// TwinCAT 3 PLC project tesimplc
// ProgramVersion: 3.1.0.8
// libraries:
//   Tc2_ControllerToolbox, * (Beckhoff Automation GmbH)
//   Tc2_Math, * (Beckhoff Automation GmbH)
//   Tc2_ModbusSrv, * (Beckhoff Automation GmbH)
//   Tc2_Standard, * (Beckhoff Automation GmbH)
//   Tc2_System, * (Beckhoff Automation GmbH)
//   Tc2_TcpIp, * (Beckhoff Automation GmbH)
//   Tc2_Utilities, * (Beckhoff Automation GmbH)
//   Tc3_Interfaces, * (Beckhoff Automation GmbH)
//   Tc3_Module, * (Beckhoff Automation GmbH)
// project tree:
//   DUTs/ MODBUS_DATA_MAP.TcDUT, XMEAS_IDX.TcDUT, XMEAS_IO_IDX.TcDUT, XMEAS_MBS_IDX.TcDUT, XMV_IDX.TcDUT, XMV_IO_IDX.TcDUT
//   funcs/ adc_to_float_pv.TcPOU (not stored), pv_float_to_dac.TcPOU
//   / GlobalTextList.TcGTLO, MainTask.TcTTO, Visualization Manager.TcVMO (not stored), VISU_TASK.TcTTO
//   GVLs/ GVL_NAMES.TcGVL, G_ICAL.TcGVL, G_IO.TcGVL, G_PARAMS.TcGVL
//   POUs/FBModbus/ FB_mb_to_val.TcPOU, FB_ModbusPoll.TcPOU, FB_ReadModbus.TcPOU, FB_HexStringToReal.TcPOU
//   POUs/FBUtils/ FB_CSV_Writer.TcPOU, FB_LFSR.TcPOU, FB_recursiveFilter.TcPOU
//   POUs/FB_Networks/ FB_NoNet.TcPOU
//   POUs/FB_Networks/iMesh/ FB_3eTI_iMesh_Base.TcPOU, FB_3eTI_iMesh_Cal.TcPOU, FB_3eTI_iMesh_GasSensor.TcPOU, FB_3eTI_iMesh_LFSR.TcPOU, FB_3eTI_iMesh_TESIM.TcPOU, FB_3eTI_TestSignals.TcPOU
//   POUs/FB_Networks/PCOneLink/ FB_PC_LFSR.TcPOU, FB_PC_OneLink_Base.TcPOU, FB_PC_OneLink_Cal.TcPOU, FB_PC_OneLink_GasSensor.TcPOU, FB_PC_OneLink_TESIM.TcPOU, FB_PC_OneLink_TestSignals.TcPOU
//   POUs/FB_Networks/Yokogawa/ FB_Yokogawa_LFSR.TcPOU, FB_Yokogawa_TestSignals.TcPOU, FB_Yokogawa_Base.TcPOU, FB_Yokogawa_GasSensor.TcPOU
//   POUs/ MAIN_oo.TcPOU
//   VISUs/ ImagePool.TcIPO (not stored), TankView.TcVIS, TESimView.TcPOU
//   zzArchive/ MAIN_wsn.TcPOU
// real-time tasks:
//   TASK MainTask: cycle T#10ms, priority 1, ADS port 350
//   TASK VISU_TASK: cycle T#100000us, priority 30, ADS port 351
// I/O:
//   DEVICE Device 1 (EtherCAT), AmsNetId 5.20.215.224.2.1
//     Term 1 (EK1200) [EK1200-5000 EtherCAT Power supply (2A E-Bus)]
//       Term 2 (EL3058) [EL3058 8Ch. Ana. Input 4-20mA]
//       Term 3 (EL4028) [EL4028 8Ch. Ana. Output 4-20mA, 12bit]
//       Term 4 (EL1808) [EL1808 8Ch. Dig. Input 24V, 3ms]
//       Term 5 (EL2808) [EL2808 8Ch. Dig. Output 24V, 0.5A]
//       Term 6 (EL3068) [EL3068 8Ch. Ana. Input 0-10V]
//       Term 7 (EL4008) [EL4008 8Ch. Ana. Output 0-10V, 12bit]
//       Term 8 (EL9011) [EL9011 End Terminal]
// variable links:
//   tesimplc/tesimplc Instance <-> Device 1 (EtherCAT)/Term 1 (EK1200)/Term 2 (EL3058)
//     MainTask Inputs/G_IO.XMEAS_IO_IIN[{1..4}] <-> AI Standard Channel {1..4}/Value  (4 links)
//     MainTask Inputs/G_IO.XMV_IO_IIN[{1..4}] <-> AI Standard Channel {5..8}/Value  (4 links)
//   tesimplc/tesimplc Instance <-> Device 1 (EtherCAT)/Term 1 (EK1200)/Term 3 (EL4028)
//     MainTask Outputs/G_IO.XMEAS_IO_IOUT[{1..4}] <-> AO Outputs Channel {1..4}/Analog output  (4 links)
//     MainTask Outputs/G_IO.XMV_IO_IOUT[{1..4}] <-> AO Outputs Channel {5..8}/Analog output  (4 links)
//   tesimplc/tesimplc Instance <-> Device 1 (EtherCAT)/Term 1 (EK1200)/Term 7 (EL4008)
//     MainTask Outputs/G_IO.XMEAS_IO_VOUT[{1..8}] <-> AO Outputs Channel {1..8}/Analog output  (8 links)

CONFIGURATION tesimplc
    RESOURCE PLC ON TwinCAT3
        TASK MainTask(INTERVAL := T#10ms, PRIORITY := 1);
        TASK VISU_TASK(INTERVAL := T#100000us, PRIORITY := 30);
        PROGRAM MAIN_oo WITH MainTask : MAIN_oo;
        PROGRAM VisuElems_Visu_Prg WITH VISU_TASK : VisuElems.Visu_Prg;
    END_RESOURCE
END_CONFIGURATION

// ---- DUTs/MODBUS_DATA_MAP.TcDUT
TYPE MODBUS_DATA_MAP :
STRUCT
	_ipAddress : STRING;
	_startAddress : WORD;
END_STRUCT
END_TYPE

// ---- DUTs/XMEAS_IDX.TcDUT
TYPE XMEAS_IDX:	
	( 
		A_FLOW			:=1,
		D_FLOW			:=2,
		E_FLOW			:=3,
		AC_FLOW			:=4,
		P_REACTOR		:=7,
		L_REACTOR		:=8,
		T_REACTOR		:=9,
		L_SEPARATOR		:=12,
		L_STRIPPER		:=15
	);
END_TYPE

// ---- DUTs/XMEAS_IO_IDX.TcDUT
TYPE XMEAS_IO_IDX :
	( 
		A_FLOW			:=1,
		D_FLOW			:=2,
		E_FLOW			:=3,
		P_REACTOR		:=4,
		AC_FLOW			:=4
	);
END_TYPE

// ---- DUTs/XMEAS_MBS_IDX.TcDUT
TYPE XMEAS_MBS_IDX :
(
	A_FLOW			:=1,
	D_FLOW			:=2,
	E_FLOW			:=3,
	P_REACTOR		:=4,
	AC_FLOW			:=4
);
END_TYPE

// ---- DUTs/XMV_IDX.TcDUT
TYPE XMV_IDX :
(
	D_FLOW_VALVE			:=1,
	E_FLOW_VALVE			:=2,	
	A_FLOW_VALVE			:=3,
	REACTOR_CWFV			:=10
);
END_TYPE

// ---- DUTs/XMV_IO_IDX.TcDUT
TYPE XMV_IO_IDX :
(
	D_FLOW_VALVE			:=1,
	E_FLOW_VALVE			:=2,	
	A_FLOW_VALVE			:=3,
	REACTOR_CWFV			:=4
);
END_TYPE

// ---- GVLs/GVL_NAMES.TcGVL
VAR_GLOBAL
	xmv_names: ARRAY[1..12] OF STRING := [
		'D Feed',
		'E Feed',
		'A Feed',
		'A+C Feed',
		'Recycle Valve',
		'Purge Valve',
		'Separator Valve',
		'Stripper Valve',
		'Steam valve',
		'Reactor Coolant',
		'Condenser Coolant',
		'Agitator Speed' ];

	xmeas_names: ARRAY[1..41] OF STRING := [
		'A Feed (kscmh)',
		'D Feed (kg/hr)',
		'E Feed (kg/hr)',
		'A+C Feed (kscmh)',
		'Recycle Flow (kscmh)',
		'Reactor Feed (kscmh)',
		'Reactor Pressure (kPa)',
		'Reactor Level (%)',
		'Reactor Temp. (°C)',
		'Purge Rate (kscmh)',
		'Sep Temp. (°C)',
		'Sep Level (%)',
		'Sep Pressure (kPa)',
		'Sep Underflow (m³/hr)',
		'Stripper Level (%)',
		'Stripper Pressure (kPa)',
		'Stripper Underflow (m³/hr)',
		'Stripper Temp. (°C)',
		'Steam Flow (kg/hr)',
		'Compressor Work (kW)',
		'React. Cool. Temp. (°C)',
		'Cond. Cool. Temp. (°C)',
		'Feed A (mole %)',
		'Feed B (mole %)',
		'Feed C (mole %)',
		'Feed D (mole %)',
		'Feed E (mole %)',
		'Feed F (mole %)',
		'Purge     % A (mole %)',
		'Purge     % B (mole %)',
		'Purge     % C (mole %)',
		'Purge     % D (mole %)',
		'Purge     % E (mole %)',
		'Purge     % F (mole %)',
		'Purge     % G (mole %)',
		'Purge     % H (mole %)',
		'Product D (mole %)',
		'Product E (mole %)',
		'Product F (mole %)',
		'Product G (mole %)',
		'Product H (mole %)' ];
END_VAR

// ---- GVLs/G_ICAL.TcGVL
VAR_GLOBAL
	
	// represents the net DC offset compensation multiplier
	XMEAS_ILOOP_CAL	: ARRAY[1..4] OF LREAL	:= 
				[
					// XMEAS tx-rx path
					-39, // A flow
					-9, // D flow
					8, // E flow
					4  // Reactor pressure
				];		
				
	XMV_ILOOP_CAL	: ARRAY[1..4] OF LREAL	:= 
				[
					// XMV tx-rx path
					-11, 	// D valve
					-11, 	// E valve
					15, 	// A valve
					-1	 	// RCW Valve
				];					
END_VAR

// ---- GVLs/G_IO.TcGVL
VAR_GLOBAL CONSTANT
	
END_VAR

VAR_GLOBAL
	
	// specify network type
	// 100 					: ISA110.11a iMesh calibration
	// 101 					: ISA110.11a iMesh TESIM
	// 102 					: ISA110.11a iMesh test signals
	// 110					: ISA100.11a iMesh PN Sequence generation
	
	// 200 					: PhoenixContact calibration
	// 201					: PhoenixContact TESIM
	// 202					: PhoenixContact test signals
	// 210					: ISA100.11a PC OneLink PN Sequence generation
	
	NET_TYPE				:	DINT := 0;
	GO						:	BOOL := FALSE;
	MODE					:	UINT := 1;
	
	// operating time
	OPTIME					:	LREAL := 0.0;
	
	// for the current-based control solutions
	XMEAS_IO_IOUT	AT %Q*		:	ARRAY[1..4] OF INT;
	XMEAS_IO_IIN	AT %I*		:	ARRAY[1..4] OF INT;
	XMV_IO_IOUT		AT %Q*		:	ARRAY[1..4] OF INT;
	XMV_IO_IIN		AT %I*		:	ARRAY[1..4] OF INT;
	
	// for the voltage-based control solutions
	XMEAS_IO_VOUT 	AT %Q*		:	ARRAY[1..8] OF INT;
	
	// XMEAS reported by tesim
	XMEAS						:	ARRAY[1..41] OF LREAL;
	XMEAS_RX					:	ARRAY[1..41] OF LREAL;
	
	// XMEAS seen by the network
	MBS_XMEAS_RAW				:	ARRAY[1..4] OF REAL;
	MBS_XMEAS					:	ARRAY[1..4] OF REAL;
	MBS_XMEAS_CAL_OFFSET		:	ARRAY[1..4] OF REAL := [0.0215, 0.0175, 0.0195, 0.0216];

	// XMV values reported by tesim
	XMV							:	ARRAY[1..12] OF LREAL;
	XMV_RX						:	ARRAY[1..12] OF LREAL;
	
	// XMV seen by the network
	//NET_XMV_RAW						:	ARRAY[1..4] OF LREAL;
	NET_XMV							:	ARRAY[1..4] OF REAL;
	
	// setpoints
	PROD_RATE					:	LREAL;
	P_REACTOR					:	LREAL;
	L_REACTOR					:	LREAL;
	T_REACTOR					:	LREAL;
	PCT_G_SP					:	LREAL;
	L_SEPARATOR					:	LREAL;
	L_STRIPPER					:	LREAL;
	
	// filtered (smoothed) values
	P_REACTOR_SM					:	LREAL;
	
	// production metrics
	COST						:	LREAL :=0.0;
	PctG						:	LREAL :=0.0;
	
	// disturbances as set in tesim
	IDV							:	ARRAY[1..20] OF DINT;
	
	// shutdown indicator
	SD_FLAG						: 	BOOL	:= FALSE;
	
END_VAR

// ---- GVLs/G_PARAMS.TcGVL
VAR_GLOBAL
	IOUT_WD_MAX	:	INT		:=32767;
	IOUT_WD_MIN	:	INT		:=0;
	VOUT_WD_MAX	:	INT		:=32767;
	VOUT_WD_MIN	:	INT		:=0;
	
	// XMEAS RANGES
	A_FLOW_MAX 		:	LREAL	:=10.0;
	D_FLOW_MAX		:	LREAL	:=7500.0;
	E_FLOW_MAX		:	LREAL	:=7500.0;
	AC_FLOW_MAX		:	LREAL	:=50.0;
	P_REACTOR_MAX	:	LREAL	:=3000.0;
	
	A_FLOW_MIN 		:	LREAL	:=0.0;
	D_FLOW_MIN		:	LREAL	:=0.0;
	E_FLOW_MIN		:	LREAL	:=0.0;
	AC_FLOW_MIN		:	LREAL	:=0.0;
	P_REACTOR_MIN	:	LREAL	:=0.0;
	
	// XMV RANGES
	A_FLOW_VALVE_MAX	: LREAL	:=100.0;
	D_FLOW_VALVE_MAX	: LREAL	:=100.0;
	E_FLOW_VALVE_MAX	: LREAL	:=100.0;
	REACTOR_CWFV_MAX	: LREAL	:=100.0;
	
	A_FLOW_VALVE_MIN	: LREAL			:=0.0;
	D_FLOW_VALVE_MIN	: LREAL			:=0.0;
	E_FLOW_VALVE_MIN	: LREAL			:=0.0;
	REACTOR_CWFV_MIN	: LREAL			:=0.0;
	
	// Device limits
	VOUT_MAX		:	LREAL	:=10.0;
	VOUT_MIN		:	LREAL	:=0.0;
	IOUT_MAX		:	LREAL	:=20.0;
	IOUT_MIN		:	LREAL	:=4.0;
	

END_VAR

// ---- POUs/MAIN_oo.TcPOU
PROGRAM MAIN_oo
VAR
	
	// network interface/simulator function blocks
	netiMeshCal				:FB_3eTI_iMesh_Cal;
	netiMeshTESIM			:FB_3eTI_iMesh_TESIM;
	netiMeshTestSignals		:FB_3eTI_TestSignals;
	netiMeshGasSensor		:FB_3eTI_iMesh_GasSensor;
	netiMeshLFSR			:FB_3eTI_iMesh_LFSR;
	
	netPCCal				:FB_PC_OneLink_Cal;
	netPCTESIM				:FB_PC_OneLink_TESIM;
	netPCTestSignals		:FB_PC_OneLink_TestSignals;
	netPCGasSensor			:FB_PC_OneLink_GasSensor;
	netPC_LFSR				:FB_PC_LFSR;
	
	// yokogawa signals
	netYokoTestSignals		:FB_Yokogawa_TestSignals;
	netYokoLFSR				:FB_Yokogawa_LFSR;
	netYokoGasSensor		:FB_Yokogawa_GasSensor;

	netNoNet				:FB_NoNet;
	
END_VAR



CASE NET_TYPE OF 
	100:
	netiMeshCal();
	101:
	netiMeshTESIM();
	102:
	netiMeshTestSignals();
	103:
	netiMeshGasSensor();
	110:
	netiMeshLFSR();
	
	200:
	netPCCal();
	201:
	netPCTESIM();
	202:
	netPCTestSignals();
	203:
	netPCGasSensor();	
	210:
	netPC_LFSR();
	
	300:
	301:
	302:
	netYokoTestSignals();
	303:
	netYokoGasSensor();
	310:
	netYokoLFSR();
	
	
ELSE
	netnoNet();
	
END_CASE

END_PROGRAM

// ---- POUs/FB_Networks/iMesh/FB_3eTI_iMesh_Cal.TcPOU
FUNCTION_BLOCK FB_3eTI_iMesh_Cal EXTENDS FB_3eTI_TestSignals
VAR_INPUT
END_VAR
VAR_OUTPUT
END_VAR
VAR
		//common calibration variables
	cal_tm 			:	TIME := T#20S;
	cal_tm_task 	:	TIME := T#100MS;
	cal_emode : E_CTRL_MODE := eCTRL_MODE_ACTIVE;
	cal_override	: BOOL	:= TRUE;
	cal_pv_mbs: ARRAY[1..4] OF LREAL := [0.0,0.0,0.0,0.0];
	cal_pv: ARRAY[1..4] OF LREAL := [0.0,0.0,0.0,0.0];
		
	// moving average
	cal_mva_work:	ARRAY[1..4] OF ARRAY[1..cal_mva_nWorkArray_SIZEOF] OF LREAL;
	cal_mva_st	:   ARRAY[1..4] OF ST_CTRL_MOVING_AVERAGE_PARAMS := [
		(	tTaskCycleTime:=cal_tm_task, 
			tCtrlCycleTime:=cal_tm,
			nSamplesToFilter:=cal_mva_nSamplesToFilter,
			nWorkArray_SIZEOF:=cal_mva_nWorkArray_SIZEOF),
		(	tTaskCycleTime:=cal_tm_task, 
			tCtrlCycleTime:=cal_tm,
			nSamplesToFilter:=cal_mva_nSamplesToFilter,
			nWorkArray_SIZEOF:=cal_mva_nWorkArray_SIZEOF),
		(	tTaskCycleTime:=cal_tm_task, 
			tCtrlCycleTime:=cal_tm,
			nSamplesToFilter:=cal_mva_nSamplesToFilter,
			nWorkArray_SIZEOF:=cal_mva_nWorkArray_SIZEOF),
		(	tTaskCycleTime:=cal_tm_task, 
			tCtrlCycleTime:=cal_tm,
			nSamplesToFilter:=cal_mva_nSamplesToFilter,
			nWorkArray_SIZEOF:=cal_mva_nWorkArray_SIZEOF)
	];
	fb_cal_mva	:	ARRAY[1..4] OF FB_CTRL_MOVING_AVERAGE := [ 
		(eMode:=cal_emode), 
		(eMode:=cal_emode), 
		(eMode:=cal_emode), 
		(eMode:=cal_emode)];
	cal_mva_mbs :	ARRAY[1..4] OF LREAL;

	// more common cal vars		
	cal_10v_dcoffset: ARRAY[1..4] OF LREAL;
	cal_ii: INT;
	cal_diff: ARRAY[1..4] OF LREAL;
	cal_frac: ARRAY[1..4] OF LREAL;
	
END_VAR
VAR CONSTANT
	cal_mva_nSamplesToFilter : UINT := 40;
	cal_mva_nWorkArray_SIZEOF: UINT := 400;
END_VAR


// call the base class to query test signal values
SUPER^();

// CALIBRATION SECTION
IF cal_override THEN
	FOR cal_ii := 1 TO 4 DO
		CASE cal_ii OF
			1:
			G_IO.XMEAS[XMEAS_IDX.A_FLOW]:=0.5;
			2:
			G_IO.XMEAS[XMEAS_IDX.D_FLOW] := 1500;
			3:
			G_IO.XMEAS[XMEAS_IDX.E_FLOW] := 1500;
			4:
			G_IO.XMEAS[XMEAS_IDX.AC_FLOW] := 2500;
		END_CASE
	END_FOR
END_IF
IF cal_emode=eCTRL_MODE_ACTIVE THEN
	FOR cal_ii := 1 TO 4 DO
		CASE cal_ii OF
			1:
			cal_pv_mbs[cal_ii] := G_IO.MBS_XMEAS[XMEAS_MBS_IDX.A_FLOW];
			cal_pv[cal_ii] := G_IO.XMEAS[XMEAS_IDX.A_FLOW];
			2:
			cal_pv_mbs[cal_ii] := G_IO.MBS_XMEAS[XMEAS_MBS_IDX.D_FLOW];
			cal_pv[cal_ii] := G_IO.XMEAS[XMEAS_IDX.D_FLOW];
			3:
			cal_pv_mbs[cal_ii] := G_IO.MBS_XMEAS[XMEAS_MBS_IDX.E_FLOW];
			cal_pv[cal_ii] := G_IO.XMEAS[XMEAS_IDX.E_FLOW];
			4:
			cal_pv_mbs[cal_ii] := G_IO.MBS_XMEAS[XMEAS_MBS_IDX.AC_FLOW];
			cal_pv[cal_ii] := G_IO.XMEAS[XMEAS_IDX.AC_FLOW];
		END_CASE
	
		// calculate moving average
		cal_mva_st[cal_ii].pWorkArray_ADR	:= ADR(cal_mva_work[cal_ii]);
		fb_cal_mva[cal_ii].fIn := cal_pv_mbs[cal_ii];
		fb_cal_mva[cal_ii](stParams:=cal_mva_st[cal_ii], eMode:=cal_emode);
		cal_mva_mbs[cal_ii] := fb_cal_mva[cal_ii].fOut;	
		
		// calculate dc offset
		IF ABS(cal_pv[cal_ii]) > 0.0 THEN
			cal_diff[cal_ii]:=cal_mva_mbs[cal_ii]-cal_pv[cal_ii];
			cal_frac[cal_ii]:=cal_diff[cal_ii]/cal_pv[cal_ii];
			cal_10v_dcoffset[cal_ii] := 10.0*cal_frac[cal_ii];
		END_IF
		
	END_FOR	
END_IF

END_FUNCTION_BLOCK

// ---- POUs/FB_Networks/iMesh/FB_3eTI_TestSignals.TcPOU
FUNCTION_BLOCK FB_3eTI_TestSignals EXTENDS FB_3eTI_iMesh_Base
VAR_INPUT
END_VAR
VAR_OUTPUT
END_VAR
VAR
END_VAR


G_PARAMS.A_FLOW_MAX 		:=10.0;
G_PARAMS.D_FLOW_MAX			:=10.0;
G_PARAMS.E_FLOW_MAX			:=10.0;
G_PARAMS.AC_FLOW_MAX		:=10.0;

G_PARAMS.A_FLOW_MIN 		:=0.0;
G_PARAMS.D_FLOW_MIN			:=0.0;
G_PARAMS.E_FLOW_MIN			:=0.0;
G_PARAMS.AC_FLOW_MIN		:=0.0;

// execute the signal conversion
SUPER^();

END_FUNCTION_BLOCK

// ---- POUs/FB_Networks/iMesh/FB_3eTI_iMesh_Base.TcPOU
FUNCTION_BLOCK FB_3eTI_iMesh_Base
VAR_INPUT
	
	// THIS IS FOR THE ISA100.11A GATEWAY
	mbAddrs : ARRAY[1..4] OF MODBUS_DATA_MAP :=  [ 
			(_ipAddress := '192.168.254.253', _startAddress:= 6), 
			(_ipAddress := '192.168.254.253', _startAddress:= 18),
			(_ipAddress := '192.168.254.253', _startAddress:= 30),
			(_ipAddress := '192.168.254.253', _startAddress:= 42)
		];
		
END_VAR

VAR
	fbReadMB 	: FB_ReadModbus;
	ii			: INT:=0;
END_VAR

VAR_OUTPUT
END_VAR

VAR
END_VAR

//
// BEGIN PRODUCE THE DATA
//
// XMEAS values will come from the external TESIM program using ADS

// VOLTAGES
XMEAS_IO_VOUT[XMEAS_IO_IDX.A_FLOW]		:= pv_float_to_dac(pv:=XMEAS[XMEAS_IDX.A_FLOW],		pv_max:=G_PARAMS.A_FLOW_MAX, pv_min:=G_PARAMS.A_FLOW_MIN, dac_max:=VOUT_WD_MAX, dac_min:=0);
XMEAS_IO_VOUT[XMEAS_IO_IDX.D_FLOW]		:= pv_float_to_dac(pv:=XMEAS[XMEAS_IDX.D_FLOW],		pv_max:=G_PARAMS.D_FLOW_MAX, pv_min:=G_PARAMS.D_FLOW_MIN, dac_max:=VOUT_WD_MAX, dac_min:=0);
XMEAS_IO_VOUT[XMEAS_IO_IDX.E_FLOW]		:= pv_float_to_dac(pv:=XMEAS[XMEAS_IDX.E_FLOW],		pv_max:=G_PARAMS.E_FLOW_MAX, pv_min:=G_PARAMS.E_FLOW_MIN, dac_max:=VOUT_WD_MAX, dac_min:=0);
XMEAS_IO_VOUT[XMEAS_IO_IDX.AC_FLOW]	:= pv_float_to_dac(pv:=XMEAS[XMEAS_IDX.AC_FLOW],	pv_max:=G_PARAMS.AC_FLOW_MAX, pv_min:=G_PARAMS.AC_FLOW_MIN, dac_max:=VOUT_WD_MAX, dac_min:=0);

//
// BEGIN MODBUS POLLING SEGMENT from the GATEWAY
//
fbReadMB(n:=4, addrs := ADR(mbAddrs) );

// poll modbus registers
G_IO.MBS_XMEAS_RAW[XMEAS_MBS_IDX.A_FLOW] := fbReadMB.registerValues[XMEAS_MBS_IDX.A_FLOW] + MBS_XMEAS_CAL_OFFSET[1];
G_IO.MBS_XMEAS_RAW[XMEAS_MBS_IDX.D_FLOW] := fbReadMB.registerValues[XMEAS_MBS_IDX.D_FLOW]+ MBS_XMEAS_CAL_OFFSET[2];
G_IO.MBS_XMEAS_RAW[XMEAS_MBS_IDX.E_FLOW] := fbReadMB.registerValues[XMEAS_MBS_IDX.E_FLOW] + MBS_XMEAS_CAL_OFFSET[3];
G_IO.MBS_XMEAS_RAW[XMEAS_MBS_IDX.AC_FLOW] := fbReadMB.registerValues[XMEAS_MBS_IDX.AC_FLOW] + MBS_XMEAS_CAL_OFFSET[4];

// convert raw modbus signals to process signals
G_IO.MBS_XMEAS[XMEAS_MBS_IDX.A_FLOW]	:=	LREAL_TO_REAL(adc_to_float_pv(G_IO.MBS_XMEAS_RAW[XMEAS_MBS_IDX.A_FLOW],		pv_max:=G_PARAMS.A_FLOW_MAX, 		pv_min:=G_PARAMS.A_FLOW_MIN, 	i_max:=G_PARAMS.VOUT_MAX, i_min:=G_PARAMS.VOUT_MIN));
G_IO.MBS_XMEAS[XMEAS_MBS_IDX.D_FLOW]	:=	LREAL_TO_REAL(adc_to_float_pv(G_IO.MBS_XMEAS_RAW[XMEAS_MBS_IDX.D_FLOW],		pv_max:=G_PARAMS.D_FLOW_MAX, 		pv_min:=G_PARAMS.D_FLOW_MIN, 	i_max:=G_PARAMS.VOUT_MAX, i_min:=G_PARAMS.VOUT_MIN));
G_IO.MBS_XMEAS[XMEAS_MBS_IDX.E_FLOW]	:=	LREAL_TO_REAL(adc_to_float_pv(G_IO.MBS_XMEAS_RAW[XMEAS_MBS_IDX.E_FLOW],		pv_max:=G_PARAMS.E_FLOW_MAX, 		pv_min:=G_PARAMS.E_FLOW_MIN, 	i_max:=G_PARAMS.VOUT_MAX, i_min:=G_PARAMS.VOUT_MIN));
G_IO.MBS_XMEAS[XMEAS_MBS_IDX.AC_FLOW]	:=	LREAL_TO_REAL(adc_to_float_pv(G_IO.MBS_XMEAS_RAW[XMEAS_MBS_IDX.AC_FLOW],	pv_max:=G_PARAMS.AC_FLOW_MAX, 	pv_min:=G_PARAMS.AC_FLOW_MIN, i_max:=G_PARAMS.VOUT_MAX, i_min:=G_PARAMS.VOUT_MIN));

// capture the received state of XMEAS
FOR ii := 1 TO 41 DO
	XMEAS_RX[ii]:=XMEAS[ii];
END_FOR
XMEAS_RX[XMEAS_IDX.A_FLOW] := G_IO.MBS_XMEAS[XMEAS_MBS_IDX.A_FLOW];
XMEAS_RX[XMEAS_IDX.D_FLOW] := G_IO.MBS_XMEAS[XMEAS_MBS_IDX.D_FLOW];
XMEAS_RX[XMEAS_IDX.E_FLOW] := G_IO.MBS_XMEAS[XMEAS_MBS_IDX.E_FLOW];
XMEAS_RX[XMEAS_IDX.AC_FLOW] := G_IO.MBS_XMEAS[XMEAS_MBS_IDX.AC_FLOW];

// capture the received state of XMV
FOR ii := 1 TO 12 DO
	XMV_RX[ii]:=XMV[ii];
END_FOR

//
// END MODBUS POLLING SEGMENT from the GATEWAY
//

END_FUNCTION_BLOCK

// ---- POUs/FBModbus/FB_ReadModbus.TcPOU
FUNCTION_BLOCK FB_ReadModbus

VAR_INPUT
	n			: INT; 	// number of modbus clients
	addrs 		: POINTER TO ARRAY[1..50] OF MODBUS_DATA_MAP;
	intervalToSampleData : TIME := T#1S; 	//modbus update rate (lower rate = more disk usage) default : 5 seconds
END_VAR

VAR_OUTPUT
	
	// input register values
	registerValues : ARRAY[0..50] OF REAL;
END_VAR

VAR
	addr: MODBUS_DATA_MAP;
	mb	: ARRAY[1..50] OF FB_ModbusPoll;
	
	//holds how many readings have been taken from initial download
	numberOfReadingsTaken : INT;

	ii: INT;
END_VAR


FOR ii:=1 TO n DO
	addr := addrs^[ii];
	mb[ii].ipAd := addr._ipAddress;
	mb[ii].startAddr := addr._startAddress;
	mb[ii](value => registerValues[ii]);
END_FOR

END_FUNCTION_BLOCK

// ---- POUs/FBModbus/FB_ModbusPoll.TcPOU
FUNCTION_BLOCK FB_ModbusPoll

VAR_INPUT
	ipAd : STRING; // the ip address of the modbus server
	startAddr : WORD; // the start address
END_VAR

VAR_OUTPUT
	value : REAL; //the modbus data
END_VAR

VAR
	dataStr :STRING;
	bModbusTick : BOOL;
	fbReadRegs : FB_MBReadInputRegs;
	converter : FB_HexStringToReal;
	arr : ARRAY [0..2] OF WORD;
END_VAR

//setup the modbus block
fbReadRegs.sIPAddr := ipAd; //gateway ip
fbReadRegs.nTCPPort := MODBUS_TCP_PORT; //502
fbReadRegs.nUnitID := 16#FF; //255
fbReadRegs.nQuantity := 3; //3 words
fbReadRegs.tTimeout := T#5S; //30 sec timout
fbReadRegs.nMBAddr := startAddr;
fbReadRegs.cbLength := 6;//nQuantity*2
fbReadRegs.pDestAddr := ADR(arr); //the pointer to the array

//the rising edge of the input negate the tick to create  a rising input of change :)
fbReadRegs.bExecute := (bModbusTick := NOT bModbusTick);
//fbReadRegs.bExecute := (bModbusTick := TRUE); 

//uppercase(convert first number to hex + convert second number to hex)
dataStr := F_TOUCase(CONCAT(WORD_TO_HEXSTR(arr[1],4,TRUE),WORD_TO_HEXSTR(arr[2],4,TRUE))); 
fbReadRegs();

//use converter to convert last 2 words to a fp value
converter(str := dataStr, out => value);

END_FUNCTION_BLOCK

// ---- POUs/FBModbus/FB_HexStringToReal.TcPOU
FUNCTION_BLOCK FB_HexStringToReal
VAR_INPUT
	str :STRING;
END_VAR
VAR_OUTPUT
	out : REAL;
END_VAR
VAR
holdStr : STRING := '';
binStr : STRING := '';
bin : STRING := '';	
sExponent : INT := 1;
expVal : INT;
sMantissa : STRING;
i :INT :=0;
ar : ARRAY[0..23] OF STRING;
significand : REAL;
decVal : REAL ;

mySExponent:INT;
myEVal:REAL;
myOut:REAL;
END_VAR

//converts the hex string to binary
FOR i :=1 TO 8 BY 1 DO
	holdStr := MID(str,1,i);
	
	IF holdStr = '0' THEN
		bin := '0000';
	ELSIF holdStr = '1' THEN
		bin := '0001';
	ELSIF holdStr = '2' THEN
		bin := '0010';
	ELSIF holdStr = '3' THEN
		bin := '0011';
	ELSIF holdStr = '4' THEN
		bin := '0100';
	ELSIF holdStr = '5' THEN
		bin := '0101';
	ELSIF holdStr = '6' THEN
		bin := '0110';
	ELSIF holdStr = '7' THEN
		bin := '0111';
	ELSIF holdStr = '8' THEN
		bin := '1000';
	ELSIF holdStr = '9' THEN
		bin := '1001';
	ELSIF holdStr = 'A' THEN
		bin := '1010';
	ELSIF holdStr = 'B' THEN
		bin := '1011';
	ELSIF holdStr = 'C' THEN
		bin := '1100';
	ELSIF holdStr = 'D' THEN
		bin := '1101';
	ELSIF holdStr = 'E' THEN
		bin := '1110';
	ELSIF holdStr = 'F' THEN
		bin := '1111';
	END_IF
	
	binStr := CONCAT(binStr,bin);
		
END_FOR

//takes half of the string
binStr := RIGHT(binStr,32);

//gets rid of the sign bit bc i am assuming that it is always positive
binStr := DELETE(binStr,1,1);

//convert the first 8 bits to get the exponent value and subtract 127
sExponent := STRING_TO_INT(CONCAT('2#',LEFT(binStr,8))) - 127;

//get remaining 23 mantissa bits
sMantissa := MID(binStr,23,9);

//values to divide by
decVal := 0.5;

//mantissa value
significand := 0;

//store mantissa bits in array
FOR i := 0 TO 23 BY 1 DO
	ar[i] := MID(sMantissa,1,i);
END_FOR

//get the significand by multiplying current bit by decVal then halve the decVal
FOR i:= 1 TO 23 BY 1 DO
	significand := significand + (STRING_TO_INT(ar[i])*decVal);
	decVal := decVal/2.0;
END_FOR

//manually generate the power of 2
expVal := 2;
FOR i:= 0 TO sExponent-2 BY 1 DO
	expVal := 2*expVal;
END_FOR
mySExponent := sExponent;
myEVal:=EXPT(2.0,mySExponent);
out := (significand +1) * (myEVal);

// This was Rushad's implementation which did not work for very small values
//make the output equal to the fp number which is calculated by multiplying
//the exponent by the significand + 1
//out := (significand +1) * (expVal);
RETURN;

END_FUNCTION_BLOCK

// ---- funcs/pv_float_to_dac.TcPOU
FUNCTION pv_float_to_dac : INT
VAR_INPUT
	pv			: LREAL;
	pv_max		: LREAL;
	pv_min		: LREAL;
	dac_max		: LREAL;
	dac_min		: LREAL;
END_VAR
VAR
	pv_float_to_dac_old: INT := 0;
END_VAR

IF floatisnan(pv) THEN
	pv_float_to_dac := 0;
ELSE

	IF pv > pv_max THEN
		pv := pv_max;
	END_IF
	IF pv < pv_min THEN
		pv := pv_min;
	END_IF
	pv_float_to_dac := LREAL_TO_INT(  (((dac_max-dac_min)/(pv_max-pv_min))*pv) + dac_min  );

END_IF

END_FUNCTION

// ---- POUs/FB_Networks/iMesh/FB_3eTI_iMesh_TESIM.TcPOU
FUNCTION_BLOCK FB_3eTI_iMesh_TESIM EXTENDS FB_3eTI_iMesh_Base
VAR_INPUT
END_VAR
VAR_OUTPUT
END_VAR
VAR
END_VAR



G_PARAMS.A_FLOW_MAX 		:=1.0;
G_PARAMS.D_FLOW_MAX			:=10000.0;
G_PARAMS.E_FLOW_MAX			:=10000.0;
G_PARAMS.AC_FLOW_MAX		:=500.0;
G_PARAMS.P_REACTOR_MAX		:=3000.0;

G_PARAMS.A_FLOW_MIN 		:=0.0;
G_PARAMS.D_FLOW_MIN			:=0.0;
G_PARAMS.E_FLOW_MIN			:=0.0;
G_PARAMS.AC_FLOW_MIN		:=0.0;
G_PARAMS.P_REACTOR_MIN		:=0.0;

// execute the signal conversion
SUPER^();

(*
//
// BEGIN PRODUCE THE DATA
//
// XMEAS values will come from the external TESIM program using ADS

// VOLTAGES
XMEAS_IO_VOUT[XMEAS_IO_IDX.A_FLOW]		:= pv_float_to_dac(pv:=XMEAS[XMEAS_IDX.A_FLOW],		pv_max:=G_PARAMS.A_FLOW_MAX, pv_min:=G_PARAMS.A_FLOW_MIN, dac_max:=VOUT_WD_MAX, dac_min:=0);
XMEAS_IO_VOUT[XMEAS_IO_IDX.D_FLOW]		:= pv_float_to_dac(pv:=XMEAS[XMEAS_IDX.D_FLOW],		pv_max:=G_PARAMS.D_FLOW_MAX, pv_min:=G_PARAMS.D_FLOW_MIN, dac_max:=VOUT_WD_MAX, dac_min:=0);
XMEAS_IO_VOUT[XMEAS_IO_IDX.E_FLOW]		:= pv_float_to_dac(pv:=XMEAS[XMEAS_IDX.E_FLOW],		pv_max:=G_PARAMS.E_FLOW_MAX, pv_min:=G_PARAMS.E_FLOW_MIN, dac_max:=VOUT_WD_MAX, dac_min:=0);
XMEAS_IO_VOUT[XMEAS_IO_IDX.P_REACTOR]	:= pv_float_to_dac(pv:=XMEAS[XMEAS_IDX.P_REACTOR],	pv_max:=G_PARAMS.P_REACTOR_MAX, pv_min:=G_PARAMS.P_REACTOR_MIN, dac_max:=VOUT_WD_MAX, dac_min:=0);


//
// BEGIN MODBUS POLLING SEGMENT from the GATEWAY
//
fbReadMB(addrs := mbAddrs );

// poll modbus registers
G_IO.MBS_XMEAS_RAW[XMEAS_MBS_IDX.A_FLOW] := fbReadMB.registerValues[XMEAS_MBS_IDX.A_FLOW] + MBS_XMEAS_CAL_OFFSET[1];
G_IO.MBS_XMEAS_RAW[XMEAS_MBS_IDX.D_FLOW] := fbReadMB.registerValues[XMEAS_MBS_IDX.D_FLOW]+ MBS_XMEAS_CAL_OFFSET[2];
G_IO.MBS_XMEAS_RAW[XMEAS_MBS_IDX.E_FLOW] := fbReadMB.registerValues[XMEAS_MBS_IDX.E_FLOW] + MBS_XMEAS_CAL_OFFSET[3];
G_IO.MBS_XMEAS_RAW[XMEAS_MBS_IDX.P_REACTOR] := fbReadMB.registerValues[XMEAS_MBS_IDX.P_REACTOR] + MBS_XMEAS_CAL_OFFSET[4];

// convert raw modbus signals to process signals
G_IO.MBS_XMEAS[XMEAS_MBS_IDX.A_FLOW]	:=	LREAL_TO_REAL(adc_to_float_pv(G_IO.MBS_XMEAS_RAW[XMEAS_MBS_IDX.A_FLOW],		pv_max:=G_PARAMS.A_FLOW_MAX, 		pv_min:=G_PARAMS.A_FLOW_MIN, 	i_max:=G_PARAMS.VOUT_MAX, i_min:=G_PARAMS.VOUT_MIN));
G_IO.MBS_XMEAS[XMEAS_MBS_IDX.D_FLOW]	:=	LREAL_TO_REAL(adc_to_float_pv(G_IO.MBS_XMEAS_RAW[XMEAS_MBS_IDX.D_FLOW],		pv_max:=G_PARAMS.D_FLOW_MAX, 		pv_min:=G_PARAMS.D_FLOW_MIN, 	i_max:=G_PARAMS.VOUT_MAX, i_min:=G_PARAMS.VOUT_MIN));
G_IO.MBS_XMEAS[XMEAS_MBS_IDX.E_FLOW]	:=	LREAL_TO_REAL(adc_to_float_pv(G_IO.MBS_XMEAS_RAW[XMEAS_MBS_IDX.E_FLOW],		pv_max:=G_PARAMS.E_FLOW_MAX, 		pv_min:=G_PARAMS.E_FLOW_MIN, 	i_max:=G_PARAMS.VOUT_MAX, i_min:=G_PARAMS.VOUT_MIN));
G_IO.MBS_XMEAS[XMEAS_MBS_IDX.P_REACTOR]	:=	LREAL_TO_REAL(adc_to_float_pv(G_IO.MBS_XMEAS_RAW[XMEAS_MBS_IDX.P_REACTOR],	pv_max:=G_PARAMS.P_REACTOR_MAX, 	pv_min:=G_PARAMS.P_REACTOR_MIN, i_max:=G_PARAMS.VOUT_MAX, i_min:=G_PARAMS.VOUT_MIN));


//
// END MODBUS POLLING SEGMENT from the GATEWAY
//
*)

END_FUNCTION_BLOCK

// ---- POUs/FB_Networks/iMesh/FB_3eTI_iMesh_GasSensor.TcPOU
FUNCTION_BLOCK FB_3eTI_iMesh_GasSensor EXTENDS FB_3eTI_iMesh_Base
VAR_INPUT
END_VAR
VAR_OUTPUT
END_VAR
VAR
	A 		: LREAL := 75;
	Tau 	: LREAL := 0.5;
	PV		: LREAL := 0.0;
	tk		: LREAL := 0.0;
	deltaT	:LREAL 	:= 10E-3;
	Pch     : LREAL := 10;
	remk: LREAL := 0.0;
END_VAR


// XMEAS RANGES
G_PARAMS.A_FLOW_MAX 	:=A;
G_PARAMS.D_FLOW_MAX		:=A;
G_PARAMS.E_FLOW_MAX		:=A;
G_PARAMS.AC_FLOW_MAX	:=A;

G_PARAMS.A_FLOW_MIN 	:=0.0;
G_PARAMS.D_FLOW_MIN		:=0.0;
G_PARAMS.E_FLOW_MIN		:=0.0;
G_PARAMS.AC_FLOW_MIN	:=0.0;

(* For built-in PV generator
// gas influx variables
tk := tk + deltaT;
remk := lmod(tk,2*Pch);
IF remk < Pch THEN
	PV := A*(1-EXP(-Tau*remk));
ELSE
	PV := A*EXP(-Tau*(remk-pch));
END_IF

G_IO.XMEAS[1] := PV;
G_IO.XMEAS[2] := PV;
G_IO.XMEAS[3] := PV;
G_IO.XMEAS[4] := PV;
*)

// execute the signal conversion
SUPER^();

END_FUNCTION_BLOCK

// ---- POUs/FB_Networks/iMesh/FB_3eTI_iMesh_LFSR.TcPOU
FUNCTION_BLOCK FB_3eTI_iMesh_LFSR EXTENDS FB_3eTI_iMesh_Base

VAR_INPUT
	clock_period	: TIME := T#2S;
END_VAR

VAR_OUTPUT

END_VAR

VAR
	
	level			: LREAL := 10.0;
	
	lfsr			: FB_LFSR();
	value			: LREAL :=0.0;
	jj				: INT	:= 0;
	lsfr: INT;
	
END_VAR


IF G_IO.GO THEN
		
	G_PARAMS.A_FLOW_MAX 		:=10.0;
	G_PARAMS.D_FLOW_MAX			:=10.0;
	G_PARAMS.E_FLOW_MAX			:=10.0;
	G_PARAMS.AC_FLOW_MAX		:=10.0;
	
	G_PARAMS.A_FLOW_MIN 		:=0.0;
	G_PARAMS.D_FLOW_MIN			:=0.0;
	G_PARAMS.E_FLOW_MIN			:=0.0;
	G_PARAMS.AC_FLOW_MIN		:=0.0;
	
	lfsr(gen_poly:=2#10111000, ck_period:= clock_period);
	value := level*USINT_TO_LREAL(lfsr.out);
	
	FOR jj := 1 TO 41 DO
		G_IO.XMEAS[jj] := value;
	END_FOR
	FOR jj := 1 TO 12 DO
		G_IO.XMV[jj] := value;
	END_FOR
	
	// execute the signal conversion
	SUPER^();
	
ELSE
	lfsr.reset();
END_IF

END_FUNCTION_BLOCK

// ---- POUs/FBUtils/FB_LFSR.TcPOU
FUNCTION_BLOCK FB_LFSR


VAR_INPUT
	gen_poly		: USINT := 2#10111000;
	ck_period		: TIME	:= T#5S;
END_VAR

VAR_OUTPUT
	out		:	USINT 	:= 	0;
	err		:	BOOL	:=	FALSE;
	epoch	:	USINT	:=	0;
END_VAR

VAR
	lfsr			: USINT := 16#11;  	// intial state of the LFSR
	lsb				: USINT := 0;		// output bit
	ck				: TON;
END_VAR


ck(IN:=NOT(ck.Q), PT:=ck_period);
IF ck.Q THEN
	// compute the next bit
	out := lfsr AND 16#1;
	lfsr:= SHR(lfsr,1);
	IF USINT_TO_BOOL(out) THEN
		lfsr := lfsr XOR gen_poly;
	END_IF
	// rest the timer
	ck.IN := TRUE; 
	epoch := epoch + 1;
END_IF


(*uint16_t start_state = 0xACE1u;  /* ANY nonzero start state will work. */
uint16_t lfsr = start_state;
unsigned period = 0;

    do
    {
        unsigned lsb = lfsr & 1;   /* Get LSB (i.e., the output bit). */
        lfsr >>= 1;                /* Shift register */
        if (lsb) {                 /* If the output bit is 1, apply toggle mask. */
            lfsr ^= 0xB400u;
        }
        ++period;
    } while (lfsr != start_state);

    return 0;
}

/* This: */
        if (lsb) {
            lfsr ^= 0xB400u;
        }
/* can also be written as: */
        lfsr ^= (-lsb) & 0xB400u;
/* which may produce more efficient code on some compilers */
*)

METHOD PUBLIC reset
VAR_INPUT
END_VAR
lfsr:=16#11;
out:=0;
END_METHOD

END_FUNCTION_BLOCK

// ---- POUs/FB_Networks/PCOneLink/FB_PC_OneLink_Cal.TcPOU
FUNCTION_BLOCK FB_PC_OneLink_Cal EXTENDS FB_PC_OneLink_TestSignals
VAR_INPUT
END_VAR
VAR_OUTPUT
END_VAR
VAR
END_VAR


// call the base class to query test signal values
SUPER^();

END_FUNCTION_BLOCK

// ---- POUs/FB_Networks/PCOneLink/FB_PC_OneLink_TestSignals.TcPOU
FUNCTION_BLOCK FB_PC_OneLink_TestSignals EXTENDS FB_PC_OneLink_Base
VAR_INPUT
END_VAR
VAR_OUTPUT
END_VAR
VAR
END_VAR


// XMEAS RANGES
G_PARAMS.A_FLOW_MAX 				:=10.0;
G_PARAMS.D_FLOW_MAX		:=10.0;
G_PARAMS.E_FLOW_MAX		:=10.0;
G_PARAMS.P_REACTOR_MAX	:=10.0;

G_PARAMS.A_FLOW_MIN 	:=0.0;
G_PARAMS.D_FLOW_MIN		:=0.0;
G_PARAMS.E_FLOW_MIN		:=0.0;
G_PARAMS.P_REACTOR_MIN	:=0.0;

// XMV RANGES
G_PARAMS.A_FLOW_VALVE_MAX	:=10.0;
G_PARAMS.D_FLOW_VALVE_MAX	:=10.0;
G_PARAMS.E_FLOW_VALVE_MAX	:=10.0;
G_PARAMS.REACTOR_CWFV_MAX	:=10.0;

G_PARAMS.A_FLOW_VALVE_MIN			:=0.0;
G_PARAMS.D_FLOW_VALVE_MIN			:=0.0;
G_PARAMS.E_FLOW_VALVE_MIN			:=0.0;
G_PARAMS.REACTOR_CWFV_MIN			:=0.0;

// execute the signal conversion
SUPER^();

END_FUNCTION_BLOCK

// ---- POUs/FB_Networks/PCOneLink/FB_PC_OneLink_Base.TcPOU
FUNCTION_BLOCK FB_PC_OneLink_Base
VAR_INPUT
END_VAR
VAR_OUTPUT
END_VAR
VAR
	ii: INT:=0;
	AFlowFilter: FB_recursiveFilter := (alpha := 0.3);
	DFlowFilter: FB_recursiveFilter := (alpha := 0.3);
	EFlowFilter: FB_recursiveFilter := (alpha := 0.3);
	ACFlowFilter: FB_recursiveFilter := (alpha := 0.3);
	ReactorPressureFilter: FB_recursiveFilter := (alpha := 0.0005);
END_VAR

//
// BEGIN PRODUCE THE DATA
//
// XMEAS values will come from the external TESIM program using ADS


//
// XMEAS SIGNAL PATHS
//
// CURRENT LOOPS for XMEAS Transmitters
XMEAS_IO_IOUT[XMEAS_IO_IDX.A_FLOW]		:= pv_float_to_dac(pv:=XMEAS[XMEAS_IDX.A_FLOW],		pv_max:=G_PARAMS.A_FLOW_MAX, pv_min:=G_PARAMS.A_FLOW_MIN, dac_max:=IOUT_WD_MAX, dac_min:=0);
XMEAS_IO_IOUT[XMEAS_IO_IDX.D_FLOW]		:= pv_float_to_dac(pv:=XMEAS[XMEAS_IDX.D_FLOW],		pv_max:=G_PARAMS.D_FLOW_MAX, pv_min:=G_PARAMS.D_FLOW_MIN, dac_max:=IOUT_WD_MAX, dac_min:=0);
XMEAS_IO_IOUT[XMEAS_IO_IDX.E_FLOW]		:= pv_float_to_dac(pv:=XMEAS[XMEAS_IDX.E_FLOW],		pv_max:=G_PARAMS.E_FLOW_MAX, pv_min:=G_PARAMS.E_FLOW_MIN, dac_max:=IOUT_WD_MAX, dac_min:=0);
XMEAS_IO_IOUT[XMEAS_IO_IDX.AC_FLOW]	:= pv_float_to_dac(pv:=XMEAS[XMEAS_IDX.AC_FLOW],	pv_max:=G_PARAMS.AC_FLOW_MAX, pv_min:=G_PARAMS.AC_FLOW_MIN, dac_max:=IOUT_WD_MAX, dac_min:=0);

// CURRENT LOOPS for XMEAS Receivers
G_IO.MBS_XMEAS[XMEAS_MBS_IDX.A_FLOW]	:=	LREAL_TO_REAL(adc_to_float_pv(G_IO.XMEAS_IO_IIN[XMEAS_MBS_IDX.A_FLOW]+G_ICAL.XMEAS_ILOOP_CAL[XMEAS_MBS_IDX.A_FLOW],		pv_max:=G_PARAMS.A_FLOW_MAX, 		pv_min:=G_PARAMS.A_FLOW_MIN, 	i_max:=G_PARAMS.IOUT_WD_MAX, i_min:=G_PARAMS.IOUT_WD_MIN));
G_IO.MBS_XMEAS[XMEAS_MBS_IDX.D_FLOW]	:=	LREAL_TO_REAL(adc_to_float_pv(G_IO.XMEAS_IO_IIN[XMEAS_MBS_IDX.D_FLOW]+G_ICAL.XMEAS_ILOOP_CAL[XMEAS_MBS_IDX.D_FLOW],		pv_max:=G_PARAMS.D_FLOW_MAX, 		pv_min:=G_PARAMS.D_FLOW_MIN, 	i_max:=G_PARAMS.IOUT_WD_MAX, i_min:=G_PARAMS.IOUT_WD_MIN));
G_IO.MBS_XMEAS[XMEAS_MBS_IDX.E_FLOW]	:=	LREAL_TO_REAL(adc_to_float_pv(G_IO.XMEAS_IO_IIN[XMEAS_MBS_IDX.E_FLOW]+G_ICAL.XMEAS_ILOOP_CAL[XMEAS_MBS_IDX.E_FLOW],		pv_max:=G_PARAMS.E_FLOW_MAX, 		pv_min:=G_PARAMS.E_FLOW_MIN, 	i_max:=G_PARAMS.IOUT_WD_MAX, i_min:=G_PARAMS.IOUT_WD_MIN));
G_IO.MBS_XMEAS[XMEAS_MBS_IDX.AC_FLOW]	:=	LREAL_TO_REAL(adc_to_float_pv(G_IO.XMEAS_IO_IIN[XMEAS_MBS_IDX.AC_FLOW]+G_ICAL.XMEAS_ILOOP_CAL[XMEAS_MBS_IDX.AC_FLOW],	pv_max:=G_PARAMS.AC_FLOW_MAX,   	pv_min:=G_PARAMS.AC_FLOW_MIN,   i_max:=G_PARAMS.IOUT_WD_MAX, i_min:=G_PARAMS.IOUT_WD_MIN));

// filter the noisy received values
AFlowFilter(xn:=G_IO.MBS_XMEAS[XMEAS_MBS_IDX.A_FLOW], yn=>G_IO.MBS_XMEAS[XMEAS_MBS_IDX.A_FLOW]);
DFlowFilter(xn:=G_IO.MBS_XMEAS[XMEAS_MBS_IDX.D_FLOW], yn=>G_IO.MBS_XMEAS[XMEAS_MBS_IDX.D_FLOW]);
EFlowFilter(xn:=G_IO.MBS_XMEAS[XMEAS_MBS_IDX.E_FLOW], yn=>G_IO.MBS_XMEAS[XMEAS_MBS_IDX.E_FLOW]);
ACFlowFilter(xn:=G_IO.MBS_XMEAS[XMEAS_MBS_IDX.AC_FLOW], yn=>G_IO.MBS_XMEAS[XMEAS_MBS_IDX.AC_FLOW]);

// filter the reactor pressure
ReactorPressureFilter(xn:=G_IO.XMEAS[7], yn=>G_IO.P_REACTOR_SM);

// capture the received state of XMEAS
FOR ii := 1 TO 41 DO
	XMEAS_RX[ii]:=XMEAS[ii];
END_FOR
XMEAS_RX[XMEAS_IDX.A_FLOW] := G_IO.MBS_XMEAS[XMEAS_MBS_IDX.A_FLOW];
XMEAS_RX[XMEAS_IDX.D_FLOW] := G_IO.MBS_XMEAS[XMEAS_MBS_IDX.D_FLOW];
XMEAS_RX[XMEAS_IDX.E_FLOW] := G_IO.MBS_XMEAS[XMEAS_MBS_IDX.E_FLOW];
XMEAS_RX[XMEAS_IDX.AC_FLOW] := G_IO.MBS_XMEAS[XMEAS_MBS_IDX.AC_FLOW];


//
// XMV SIGNAL PATHS
//
// CURRENT LOOPS for XMV Transmitters
XMV_IO_IOUT[XMV_IO_IDX.D_FLOW_VALVE]	:= pv_float_to_dac(pv:=XMV[XMV_IDX.D_FLOW_VALVE],	pv_max:=G_PARAMS.D_FLOW_VALVE_MAX, pv_min:=G_PARAMS.D_FLOW_VALVE_MIN, dac_max:=IOUT_WD_MAX, dac_min:=0);
XMV_IO_IOUT[XMV_IO_IDX.E_FLOW_VALVE]	:= pv_float_to_dac(pv:=XMV[XMV_IDX.E_FLOW_VALVE],	pv_max:=G_PARAMS.E_FLOW_VALVE_MAX, pv_min:=G_PARAMS.E_FLOW_VALVE_MIN, dac_max:=IOUT_WD_MAX, dac_min:=0);
XMV_IO_IOUT[XMV_IO_IDX.A_FLOW_VALVE]	:= pv_float_to_dac(pv:=XMV[XMV_IDX.A_FLOW_VALVE],	pv_max:=G_PARAMS.A_FLOW_VALVE_MAX, pv_min:=G_PARAMS.A_FLOW_VALVE_MIN, dac_max:=IOUT_WD_MAX, dac_min:=0);
XMV_IO_IOUT[XMV_IO_IDX.REACTOR_CWFV]	:= pv_float_to_dac(pv:=XMV[XMV_IDX.REACTOR_CWFV],	pv_max:=G_PARAMS.REACTOR_CWFV_MAX, pv_min:=G_PARAMS.REACTOR_CWFV_MIN, dac_max:=IOUT_WD_MAX, dac_min:=0);

// CURRENT LOOPS for XMV Receivers
G_IO.NET_XMV[XMV_IO_IDX.D_FLOW_VALVE]	:=	LREAL_TO_REAL(adc_to_float_pv(G_IO.XMV_IO_IIN[XMV_IO_IDX.D_FLOW_VALVE]+G_ICAL.XMV_ILOOP_CAL[XMV_IO_IDX.D_FLOW_VALVE],		pv_max:=G_PARAMS.D_FLOW_VALVE_MAX, 		pv_min:=G_PARAMS.D_FLOW_VALVE_MIN,	i_max:=G_PARAMS.IOUT_WD_MAX, i_min:=G_PARAMS.IOUT_WD_MIN));
G_IO.NET_XMV[XMV_IO_IDX.E_FLOW_VALVE]	:=	LREAL_TO_REAL(adc_to_float_pv(G_IO.XMV_IO_IIN[XMV_IO_IDX.E_FLOW_VALVE]+G_ICAL.XMV_ILOOP_CAL[XMV_IO_IDX.E_FLOW_VALVE],		pv_max:=G_PARAMS.E_FLOW_VALVE_MAX, 		pv_min:=G_PARAMS.E_FLOW_VALVE_MIN,	i_max:=G_PARAMS.IOUT_WD_MAX, i_min:=G_PARAMS.IOUT_WD_MIN));
G_IO.NET_XMV[XMV_IO_IDX.A_FLOW_VALVE]	:=	LREAL_TO_REAL(adc_to_float_pv(G_IO.XMV_IO_IIN[XMV_IO_IDX.A_FLOW_VALVE]+G_ICAL.XMV_ILOOP_CAL[XMV_IO_IDX.A_FLOW_VALVE],		pv_max:=G_PARAMS.A_FLOW_VALVE_MAX, 		pv_min:=G_PARAMS.A_FLOW_VALVE_MIN,	i_max:=G_PARAMS.IOUT_WD_MAX, i_min:=G_PARAMS.IOUT_WD_MIN));
G_IO.NET_XMV[XMV_IO_IDX.REACTOR_CWFV]	:=	LREAL_TO_REAL(adc_to_float_pv(G_IO.XMV_IO_IIN[XMV_IO_IDX.REACTOR_CWFV]+G_ICAL.XMV_ILOOP_CAL[XMV_IO_IDX.REACTOR_CWFV],		pv_max:=G_PARAMS.REACTOR_CWFV_MAX, 		pv_min:=G_PARAMS.REACTOR_CWFV_MIN,	i_max:=G_PARAMS.IOUT_WD_MAX, i_min:=G_PARAMS.IOUT_WD_MIN));

// capture the received state of XMV
FOR ii := 1 TO 12 DO
	XMV_RX[ii]:=XMV[ii];
END_FOR
XMV_RX[XMV_IDX.D_FLOW_VALVE] := G_IO.NET_XMV[XMV_IO_IDX.D_FLOW_VALVE];
XMV_RX[XMV_IDX.E_FLOW_VALVE] := G_IO.NET_XMV[XMV_IO_IDX.E_FLOW_VALVE];
XMV_RX[XMV_IDX.A_FLOW_VALVE] := G_IO.NET_XMV[XMV_IO_IDX.A_FLOW_VALVE];
XMV_RX[XMV_IDX.REACTOR_CWFV] := G_IO.NET_XMV[XMV_IO_IDX.REACTOR_CWFV];

END_FUNCTION_BLOCK

// ---- POUs/FBUtils/FB_recursiveFilter.TcPOU
FUNCTION_BLOCK FB_recursiveFilter

VAR_INPUT
	xn	: LREAL;
END_VAR

VAR_OUTPUT
	yn	:	LREAL;
END_VAR

VAR
	alpha:	LREAL	:= 0.025;
	yn_1 :	LREAL 	:= 0.0;
	init : 	BOOL	:= TRUE;
END_VAR


IF init THEN
	yn_1 := xn;
	init := FALSE;
END_IF
yn := alpha*xn + (1-alpha)*yn_1;
yn_1 := yn;

END_FUNCTION_BLOCK

// ---- POUs/FB_Networks/PCOneLink/FB_PC_OneLink_TESIM.TcPOU
FUNCTION_BLOCK FB_PC_OneLink_TESIM EXTENDS FB_PC_OneLink_Base
VAR_INPUT
END_VAR
VAR_OUTPUT
END_VAR
VAR
END_VAR

G_PARAMS.A_FLOW_MAX 		:=1.2;
G_PARAMS.D_FLOW_MAX			:=10000.0;
G_PARAMS.E_FLOW_MAX			:=10000.0;
G_PARAMS.AC_FLOW_MAX		:=50.0;

G_PARAMS.A_FLOW_MIN 		:=0.0;
G_PARAMS.D_FLOW_MIN			:=0.0;
G_PARAMS.E_FLOW_MIN			:=0.0;
G_PARAMS.AC_FLOW_MIN		:=0.0;

SUPER^();
(*
//
// BEGIN PRODUCE THE DATA
//
// XMEAS values will come from the external TESIM program using ADS


//
// WRITE SIGNALS to OUTPUTS
//
// CURRENT LOOPS for XMEAS Transmitters
XMEAS_IO_IOUT[XMEAS_IO_IDX.A_FLOW]		:= pv_float_to_dac(pv:=XMEAS[XMEAS_IDX.A_FLOW],		pv_max:=G_PARAMS.A_FLOW_MAX, pv_min:=G_PARAMS.A_FLOW_MIN, dac_max:=IOUT_WD_MAX, dac_min:=0);
XMEAS_IO_IOUT[XMEAS_IO_IDX.D_FLOW]		:= pv_float_to_dac(pv:=XMEAS[XMEAS_IDX.D_FLOW],		pv_max:=G_PARAMS.D_FLOW_MAX, pv_min:=G_PARAMS.D_FLOW_MIN, dac_max:=IOUT_WD_MAX, dac_min:=0);
XMEAS_IO_IOUT[XMEAS_IO_IDX.E_FLOW]		:= pv_float_to_dac(pv:=XMEAS[XMEAS_IDX.E_FLOW],		pv_max:=G_PARAMS.E_FLOW_MAX, pv_min:=G_PARAMS.E_FLOW_MIN, dac_max:=IOUT_WD_MAX, dac_min:=0);
XMEAS_IO_IOUT[XMEAS_IO_IDX.P_REACTOR]	:= pv_float_to_dac(pv:=XMEAS[XMEAS_IDX.P_REACTOR],	pv_max:=G_PARAMS.P_REACTOR_MAX, pv_min:=G_PARAMS.P_REACTOR_MIN, dac_max:=IOUT_WD_MAX, dac_min:=0);

// CURRENT LOOPS for XMV Transmitters
XMV_IO_IOUT[XMV_IO_IDX.A_FLOW_VALVE]		:= pv_float_to_dac(pv:=XMEAS[XMV_IDX.A_FLOW_VALVE],		pv_max:=G_PARAMS.A_FLOW_VALVE_MAX, pv_min:=G_PARAMS.A_FLOW_VALVE_MAX, dac_max:=IOUT_WD_MAX, dac_min:=0);
XMV_IO_IOUT[XMV_IO_IDX.D_FLOW_VALVE]		:= pv_float_to_dac(pv:=XMEAS[XMV_IDX.D_FLOW_VALVE],		pv_max:=G_PARAMS.D_FLOW_VALVE_MAX, pv_min:=G_PARAMS.D_FLOW_VALVE_MAX, dac_max:=IOUT_WD_MAX, dac_min:=0);
XMV_IO_IOUT[XMV_IO_IDX.E_FLOW_VALVE]		:= pv_float_to_dac(pv:=XMEAS[XMV_IDX.E_FLOW_VALVE],		pv_max:=G_PARAMS.E_FLOW_VALVE_MAX, pv_min:=G_PARAMS.E_FLOW_VALVE_MAX, dac_max:=IOUT_WD_MAX, dac_min:=0);
XMV_IO_IOUT[XMV_IO_IDX.REACTOR_CWFV]	:= pv_float_to_dac(pv:=XMEAS[XMV_IDX.REACTOR_CWFV],	pv_max:=G_PARAMS.REACTOR_CWFV_MAX, pv_min:=G_PARAMS.REACTOR_CWFV_MIN, dac_max:=IOUT_WD_MAX, dac_min:=0);

//
// READ SIGNALS from INPUTS
//
// CURRENT LOOPS for XMEAS Receivers
G_IO.MBS_XMEAS[XMEAS_MBS_IDX.A_FLOW]	:=	LREAL_TO_REAL(adc_to_float_pv(G_IO.XMEAS_IO_IIN[XMEAS_MBS_IDX.A_FLOW],		pv_max:=G_PARAMS.A_FLOW_MAX, 		pv_min:=G_PARAMS.A_FLOW_MIN, 	i_max:=G_PARAMS.IOUT_MAX, i_min:=G_PARAMS.IOUT_MIN));
G_IO.MBS_XMEAS[XMEAS_MBS_IDX.D_FLOW]	:=	LREAL_TO_REAL(adc_to_float_pv(G_IO.XMEAS_IO_IIN[XMEAS_MBS_IDX.D_FLOW],		pv_max:=G_PARAMS.D_FLOW_MAX, 		pv_min:=G_PARAMS.D_FLOW_MIN, 	i_max:=G_PARAMS.IOUT_MAX, i_min:=G_PARAMS.IOUT_MIN));
G_IO.MBS_XMEAS[XMEAS_MBS_IDX.E_FLOW]	:=	LREAL_TO_REAL(adc_to_float_pv(G_IO.XMEAS_IO_IIN[XMEAS_MBS_IDX.E_FLOW],		pv_max:=G_PARAMS.E_FLOW_MAX, 		pv_min:=G_PARAMS.E_FLOW_MIN, 	i_max:=G_PARAMS.IOUT_MAX, i_min:=G_PARAMS.IOUT_MIN));
G_IO.MBS_XMEAS[XMEAS_MBS_IDX.P_REACTOR]	:=	LREAL_TO_REAL(adc_to_float_pv(G_IO.XMEAS_IO_IIN[XMEAS_MBS_IDX.P_REACTOR],	pv_max:=G_PARAMS.P_REACTOR_MAX, 	pv_min:=G_PARAMS.P_REACTOR_MIN, i_max:=G_PARAMS.IOUT_MAX, i_min:=G_PARAMS.IOUT_MIN));

// CURRENT LOOPS for XMV Receivers
G_IO.NET_XMV[XMV_IO_IDX.A_FLOW_VALVE]	:=	LREAL_TO_REAL(adc_to_float_pv(G_IO.NET_XMV_RAW[XMV_IO_IDX.A_FLOW_VALVE],		pv_max:=G_PARAMS.A_FLOW_VALVE_MAX, 		pv_min:=G_PARAMS.A_FLOW_VALVE_MIN,	i_max:=G_PARAMS.IOUT_MAX, i_min:=G_PARAMS.IOUT_MIN));
G_IO.NET_XMV[XMV_IO_IDX.D_FLOW_VALVE]	:=	LREAL_TO_REAL(adc_to_float_pv(G_IO.NET_XMV_RAW[XMV_IO_IDX.D_FLOW_VALVE],		pv_max:=G_PARAMS.D_FLOW_VALVE_MAX, 		pv_min:=G_PARAMS.D_FLOW_VALVE_MIN,	i_max:=G_PARAMS.IOUT_MAX, i_min:=G_PARAMS.IOUT_MIN));
G_IO.NET_XMV[XMV_IO_IDX.E_FLOW_VALVE]	:=	LREAL_TO_REAL(adc_to_float_pv(G_IO.NET_XMV_RAW[XMV_IO_IDX.E_FLOW_VALVE],		pv_max:=G_PARAMS.E_FLOW_VALVE_MAX, 		pv_min:=G_PARAMS.E_FLOW_VALVE_MIN,	i_max:=G_PARAMS.IOUT_MAX, i_min:=G_PARAMS.IOUT_MIN));
G_IO.NET_XMV[XMV_IO_IDX.REACTOR_CWFV]	:=	LREAL_TO_REAL(adc_to_float_pv(G_IO.NET_XMV_RAW[XMV_IO_IDX.REACTOR_CWFV],		pv_max:=G_PARAMS.REACTOR_CWFV_MAX, 		pv_min:=G_PARAMS.REACTOR_CWFV_MIN,	i_max:=G_PARAMS.IOUT_MAX, i_min:=G_PARAMS.IOUT_MIN));
*)

END_FUNCTION_BLOCK

// ---- POUs/FB_Networks/PCOneLink/FB_PC_OneLink_GasSensor.TcPOU
FUNCTION_BLOCK FB_PC_OneLink_GasSensor EXTENDS FB_PC_OneLink_Base
VAR_INPUT
END_VAR
VAR_OUTPUT
END_VAR
VAR
END_VAR


// XMEAS RANGES
G_PARAMS.A_FLOW_MAX 	:=20.0;
G_PARAMS.D_FLOW_MAX		:=20.0;

G_PARAMS.A_FLOW_MIN 	:=0.0;
G_PARAMS.D_FLOW_MIN		:=0.0;

// execute the signal conversion
SUPER^();

END_FUNCTION_BLOCK

// ---- POUs/FB_Networks/PCOneLink/FB_PC_LFSR.TcPOU
FUNCTION_BLOCK FB_PC_LFSR EXTENDS FB_PC_OneLink_TestSignals

VAR_INPUT
END_VAR

VAR_OUTPUT

END_VAR

VAR
	level			: LREAL := 10.0;
	
	lfsr			: FB_LFSR;
	value			: LREAL :=0.0;
	jj				: INT	:= 0;
END_VAR


lfsr(gen_poly:=2#10111000);
value := level*USINT_TO_LREAL(lfsr.out);

FOR jj := 1 TO 41 DO
	G_IO.XMEAS[jj] := value;
END_FOR
FOR jj := 1 TO 12 DO
	G_IO.XMV[jj] := value;
END_FOR

SUPER^();

END_FUNCTION_BLOCK

// ---- POUs/FB_Networks/Yokogawa/FB_Yokogawa_TestSignals.TcPOU
FUNCTION_BLOCK FB_Yokogawa_TestSignals EXTENDS FB_Yokogawa_Base
VAR_INPUT
END_VAR
VAR_OUTPUT
END_VAR
VAR
END_VAR


G_PARAMS.A_FLOW_MAX 		:=100.0;
G_PARAMS.D_FLOW_MAX			:=100.0;
G_PARAMS.E_FLOW_MAX			:=100.0;
G_PARAMS.AC_FLOW_MAX		:=100.0;

G_PARAMS.A_FLOW_MIN 		:=0.0;
G_PARAMS.D_FLOW_MIN			:=0.0;
G_PARAMS.E_FLOW_MIN			:=0.0;
G_PARAMS.AC_FLOW_MIN		:=0.0;

(*G_IO.XMEAS[1]:=100;
G_IO.XMEAS[2]:=100;
G_IO.XMEAS[3]:=100;
G_IO.XMEAS[4]:=100;*)

// execute the signal conversion
SUPER^();

END_FUNCTION_BLOCK

// ---- POUs/FB_Networks/Yokogawa/FB_Yokogawa_Base.TcPOU
FUNCTION_BLOCK FB_Yokogawa_Base
VAR_INPUT
	
	// THIS IS FOR THE ISA100.11A GATEWAY
	mbAddrs : ARRAY[0..4] OF MODBUS_DATA_MAP :=  [ 
			(_ipAddress := '192.168.0.101', _startAddress:= 674), 
			(_ipAddress := '192.168.0.101', _startAddress:= 677),
			(_ipAddress := '192.168.0.101', _startAddress:= 680),
			(_ipAddress := '192.168.0.101', _startAddress:= 683),
			(_ipAddress := '192.168.0.101', _startAddress:= 577)
		];
		
END_VAR

VAR
	fbReadMB 	: FB_ReadModbus;
	ii			: INT:=0;
END_VAR

VAR_OUTPUT
END_VAR

VAR
END_VAR

//
// BEGIN PRODUCE THE DATA
//
// XMEAS values will come from the external TESIM program using ADS

// VOLTAGES
XMEAS_IO_IOUT[XMEAS_IO_IDX.A_FLOW]		:= pv_float_to_dac(pv:=XMEAS[XMEAS_IDX.A_FLOW],		pv_max:=G_PARAMS.A_FLOW_MAX, pv_min:=G_PARAMS.A_FLOW_MIN, dac_max:=VOUT_WD_MAX, dac_min:=0);
XMEAS_IO_IOUT[XMEAS_IO_IDX.D_FLOW]		:= pv_float_to_dac(pv:=XMEAS[XMEAS_IDX.D_FLOW],		pv_max:=G_PARAMS.D_FLOW_MAX, pv_min:=G_PARAMS.D_FLOW_MIN, dac_max:=VOUT_WD_MAX, dac_min:=0);
XMEAS_IO_IOUT[XMEAS_IO_IDX.E_FLOW]		:= pv_float_to_dac(pv:=XMEAS[XMEAS_IDX.E_FLOW],		pv_max:=G_PARAMS.E_FLOW_MAX, pv_min:=G_PARAMS.E_FLOW_MIN, dac_max:=VOUT_WD_MAX, dac_min:=0);
XMEAS_IO_IOUT[XMEAS_IO_IDX.AC_FLOW]	:= pv_float_to_dac(pv:=XMEAS[XMEAS_IDX.AC_FLOW],	pv_max:=G_PARAMS.AC_FLOW_MAX, pv_min:=G_PARAMS.AC_FLOW_MIN, dac_max:=VOUT_WD_MAX, dac_min:=0);

//
// BEGIN MODBUS POLLING SEGMENT from the GATEWAY
//
fbReadMB(n := 5, addrs := ADR(mbAddrs) );

// poll modbus registers
G_IO.MBS_XMEAS_RAW[XMEAS_MBS_IDX.A_FLOW] := fbReadMB.registerValues[XMEAS_MBS_IDX.A_FLOW] ;
G_IO.MBS_XMEAS_RAW[XMEAS_MBS_IDX.D_FLOW] := fbReadMB.registerValues[XMEAS_MBS_IDX.D_FLOW];
G_IO.MBS_XMEAS_RAW[XMEAS_MBS_IDX.E_FLOW] := fbReadMB.registerValues[XMEAS_MBS_IDX.E_FLOW];
G_IO.MBS_XMEAS_RAW[XMEAS_MBS_IDX.AC_FLOW] := fbReadMB.registerValues[XMEAS_MBS_IDX.AC_FLOW];

// convert raw modbus signals to process signals
G_IO.MBS_XMEAS[XMEAS_MBS_IDX.A_FLOW]	:=	LREAL_TO_REAL(G_IO.MBS_XMEAS_RAW[XMEAS_MBS_IDX.A_FLOW]);
G_IO.MBS_XMEAS[XMEAS_MBS_IDX.D_FLOW]	:=	LREAL_TO_REAL(G_IO.MBS_XMEAS_RAW[XMEAS_MBS_IDX.D_FLOW]);
G_IO.MBS_XMEAS[XMEAS_MBS_IDX.E_FLOW]	:=	LREAL_TO_REAL(G_IO.MBS_XMEAS_RAW[XMEAS_MBS_IDX.E_FLOW]);
G_IO.MBS_XMEAS[XMEAS_MBS_IDX.AC_FLOW]	:=	LREAL_TO_REAL(G_IO.MBS_XMEAS_RAW[XMEAS_MBS_IDX.AC_FLOW]);

// capture the received state of XMEAS
FOR ii := 1 TO 41 DO
	XMEAS_RX[ii]:=XMEAS[ii];
END_FOR
XMEAS_RX[XMEAS_IDX.A_FLOW] := G_IO.MBS_XMEAS[XMEAS_MBS_IDX.A_FLOW];
XMEAS_RX[XMEAS_IDX.D_FLOW] := G_IO.MBS_XMEAS[XMEAS_MBS_IDX.D_FLOW];
XMEAS_RX[XMEAS_IDX.E_FLOW] := G_IO.MBS_XMEAS[XMEAS_MBS_IDX.E_FLOW];
XMEAS_RX[XMEAS_IDX.AC_FLOW] := G_IO.MBS_XMEAS[XMEAS_MBS_IDX.AC_FLOW];


//
// END MODBUS POLLING SEGMENT from the GATEWAY
//

END_FUNCTION_BLOCK

// ---- POUs/FB_Networks/Yokogawa/FB_Yokogawa_LFSR.TcPOU
FUNCTION_BLOCK FB_Yokogawa_LFSR EXTENDS FB_Yokogawa_Base

VAR_INPUT
	clock_period	: TIME := T#2S;
END_VAR

VAR_OUTPUT

END_VAR

VAR
	
	level			: LREAL := 1.0;
	
	lfsr			: FB_LFSR();
	value			: LREAL :=0.0;
	jj				: INT	:= 0;
	lsfr: INT;
	
END_VAR


VAR CONSTANT
	NXMEAS: INT := 4;
	NXMV: INT := 0;
END_VAR


IF G_IO.GO THEN
		
	G_PARAMS.A_FLOW_MAX 		:=1.0;
	G_PARAMS.D_FLOW_MAX			:=1.0;
	G_PARAMS.E_FLOW_MAX			:=1.0;
	G_PARAMS.AC_FLOW_MAX		:=1.0;
	
	G_PARAMS.A_FLOW_MIN 		:=0.0;
	G_PARAMS.D_FLOW_MIN			:=0.0;
	G_PARAMS.E_FLOW_MIN			:=0.0;
	G_PARAMS.AC_FLOW_MIN		:=0.0;
	
	lfsr(gen_poly:=2#10111000, ck_period:= clock_period);
	value := level*USINT_TO_LREAL(lfsr.out);
	
	FOR jj := 1 TO NXMEAS DO
		G_IO.XMEAS[jj] := value;
	END_FOR
	FOR jj := 1 TO NXMV DO
		G_IO.XMV[jj] := value;
	END_FOR
	
	// execute the signal conversion
	SUPER^();
	
ELSE
	lfsr.reset();
END_IF

END_FUNCTION_BLOCK

// ---- POUs/FB_Networks/Yokogawa/FB_Yokogawa_GasSensor.TcPOU
FUNCTION_BLOCK FB_Yokogawa_GasSensor EXTENDS FB_Yokogawa_Base
VAR_INPUT
END_VAR
VAR_OUTPUT
END_VAR
VAR
	PVfs	: LREAL := 100.0;
	A 		: LREAL := 75.0;
	Tau 	: LREAL := 0.5;
	PV		: LREAL := 0.0;
	tk		: LREAL := 0.0;
	deltaT	:LREAL 	:= 10E-3;
	Pch     : LREAL := 10;
	remk: LREAL := 0.0;
END_VAR


// XMEAS RANGES
G_PARAMS.A_FLOW_MAX 	:=PVfs;
G_PARAMS.D_FLOW_MAX		:=PVfs;
G_PARAMS.E_FLOW_MAX		:=PVfs;
G_PARAMS.AC_FLOW_MAX	:=PVfs;

G_PARAMS.A_FLOW_MIN 	:=0.0;
G_PARAMS.D_FLOW_MIN		:=0.0;
G_PARAMS.E_FLOW_MIN		:=0.0;
G_PARAMS.AC_FLOW_MIN	:=0.0;

(* For built-in PV generator
// gas influx variables
tk := tk + deltaT;
remk := lmod(tk,2*Pch);
IF remk < Pch THEN
	PV := A*(1-EXP(-Tau*remk));
ELSE
	PV := A*EXP(-Tau*(remk-pch));
END_IF

G_IO.XMEAS[1] := PV;
G_IO.XMEAS[2] := PV;
G_IO.XMEAS[3] := PV;
G_IO.XMEAS[4] := PV;
*)

// execute the signal conversion
SUPER^();

END_FUNCTION_BLOCK

// ---- POUs/FB_Networks/FB_NoNet.TcPOU
FUNCTION_BLOCK FB_NoNet
VAR_INPUT
END_VAR
VAR_OUTPUT
END_VAR
VAR
END_VAR

END_FUNCTION_BLOCK

// ---- POUs/FBModbus/FB_mb_to_val.TcPOU
FUNCTION_BLOCK FB_mb_to_val
VAR_INPUT
	xi: REAL:=0;
	i_hi: REAL:=20.0;
	y_h: REAL:= 0.0;
END_VAR

VAR_OUTPUT
	y: REAL;
END_VAR

VAR
	xi_cal: REAL;
END_VAR



y:=y_h*xi/i_hi;
IF y>y_h THEN
	y:=y_h;
ELSIF y < 0 THEN
	y:=0.0;	
END_IF

END_FUNCTION_BLOCK

// ---- POUs/FBUtils/FB_CSV_Writer.TcPOU
FUNCTION_BLOCK FB_CSV_Writer //Matt
VAR_INPUT
	bWriteLine:	BOOL; //true if you want to write to the file
	sFileName:	STRING; //name of the file to write
	fDataPoint1:	REAL; //data point 1
	fDataPoint2:	REAL; //data point 2
END_VAR
VAR_OUTPUT
	bBusy:	BOOL;
	bError:	BOOL;
	sError:	STRING;
END_VAR
VAR
	fbFileOpen:	FB_FileOpen; //fb to open the file to begin appending
	fbFilePuts:	FB_FilePuts; //fb to write to the file
	fbFileClose: FB_FileClose; // closes the file
	
	rtWrite:	R_TRIG; //trigger
	
	nState:	INT; //state to cycle to parts of appending
	sTempPathName:	STRING; 
	sDataString:	STRING; //string to write
END_VAR

rtWrite(CLK := bWriteLine);

CASE nState OF
	0:	(*IDLE*)
		bBusy := FALSE;
		IF rtWrite.Q THEN
			sTempPathName := CONCAT(CONCAT('C:\Temp\',sFileName),'.csv');
			sDataString := CONCAT(CONCAT(CONCAT(REAL_TO_STRING(fDataPoint1),','),REAL_TO_STRING(fDataPoint2)),'$N'); 
			bBusy := TRUE;
			bError := FALSE;
			sError := '';
			nState := nState + 10;
		END_IF		
	
	10:	(*Open File*)	
		fbFileOpen(	sPathName := sTempPathName,nMode := FOPEN_MODEAPPEND,bExecute := TRUE,tTimeOut := T#1S);
		IF NOT fbFileOpen.bBusy THEN
			fbFileOpen(	bExecute := FALSE);
			IF fbFileOpen.bError THEN
				bError := TRUE;
				sError := 'Could Not Open File';
				nState := 0;
			ELSE
				nState := nState + 10;
			END_IF
		END_IF
		
	20:	(*Write Line To File*)
		fbFilePuts(	hFile := fbFileOpen.hFile,sLine := sDataString,bExecute := TRUE,tTimeout := T#1S);
		IF NOT fbFilePuts.bBusy THEN
			fbFilePuts(	bExecute := FALSE);
			IF fbFilePuts.bError THEN
				bError := TRUE;
				sError := 'Could not write to file';
				nState := nState + 10;
			ELSE
				nState := nState + 10;
			END_IF
		END_IF
		
	30:	(*Close File*)
		fbFileClose(hFile := fbFileOpen.hFile,bExecute := TRUE,tTimeout := T#1S);
		IF NOT fbFileClose.bBusy THEN
			fbFileClose(	bExecute := FALSE);
			IF fbFileClose.bError THEN
				bError := TRUE;
				sError := 'Could not close file';
				nState := 0;
			ELSE
				nState := 0;
			END_IF
		END_IF
END_CASE

END_FUNCTION_BLOCK

// ---- VISUs/TESimView.TcPOU
PROGRAM TESimView
VAR
	XMEAS_PurgeAnalyzer		:	ARRAY[1..8] OF REAL;
	XMEAS_FeedAnalyzer		:	ARRAY[1..6] OF REAL;
	XMEAS_ProductAnalyzer	:	ARRAY[1..5] OF REAL;
	i: INT := 0;	
	
XMV_STRINGS					:	ARRAY[1..12] OF WSTRING := [
									"D feed flow",
									"E feed flow", 
									"A feed flow",
									"A and C feed flow",
									"Compressor recycle valve",
									"Purpc valve",
									"Separator pot liquid flow",
									"Stripper liquid flow",
									"Stripper steam flow",
									"Reactor cooling water flow",
									"Condensor cooling water flow",
									"Agitator speed"];	
END_VAR

FOR i :=1 TO 8 DO
	XMEAS_PurgeAnalyzer[i] := G_IO.XMEAS[i+28];
END_FOR

FOR i :=1 TO 6 DO
	XMEAS_FeedAnalyzer[i] := G_IO.XMEAS[i+22];
END_FOR

FOR i :=1 TO 5 DO
	XMEAS_ProductAnalyzer[i] := G_IO.XMEAS[i+36];
END_FOR

END_PROGRAM

// ---- zzArchive/MAIN_wsn.TcPOU
PROGRAM MAIN_wsn
VAR

	fbReadMB : FB_ReadModbus;
	

	// THIS IS FOR THE WIHART GATEWAY
	//mbAddrs : ARRAY[0..1] OF MODBUS_DATA_MAP :=  [ (_ipAddress := '192.168.1.101', _startAddress:= 0), (_ipAddress := '192.168.1.101', _startAddress:= 12) ];
	
	// THIS IS FOR THE ISA100.11A GATEWAY
	mbAddrs : ARRAY[0..3] OF MODBUS_DATA_MAP :=  [ 
			(_ipAddress := '192.168.254.253', _startAddress:= 6), 
			(_ipAddress := '192.168.254.253', _startAddress:= 18),
			(_ipAddress := '192.168.254.253', _startAddress:= 30),
			(_ipAddress := '192.168.254.253', _startAddress:= 42)
		];
 
	test_input: BOOL := FALSE;
	
	//common calibration variables
	cal_tm 			:	TIME := T#20S;
	cal_tm_task 	:	TIME := T#100MS;
	cal_emode : E_CTRL_MODE := eCTRL_MODE_ACTIVE;
	cal_override	: BOOL	:= FALSE;
	cal_pv_mbs: ARRAY[1..4] OF LREAL := [0.0,0.0,0.0,0.0];
	cal_pv: ARRAY[1..4] OF LREAL := [0.0,0.0,0.0,0.0];
		
	// moving average
	cal_mva_work:	ARRAY[1..4] OF ARRAY[1..cal_mva_nWorkArray_SIZEOF] OF LREAL;
	cal_mva_st	:   ARRAY[1..4] OF ST_CTRL_MOVING_AVERAGE_PARAMS := [
		(	tTaskCycleTime:=cal_tm_task, 
			tCtrlCycleTime:=cal_tm,
			nSamplesToFilter:=cal_mva_nSamplesToFilter,
			nWorkArray_SIZEOF:=cal_mva_nWorkArray_SIZEOF),
		(	tTaskCycleTime:=cal_tm_task, 
			tCtrlCycleTime:=cal_tm,
			nSamplesToFilter:=cal_mva_nSamplesToFilter,
			nWorkArray_SIZEOF:=cal_mva_nWorkArray_SIZEOF),
		(	tTaskCycleTime:=cal_tm_task, 
			tCtrlCycleTime:=cal_tm,
			nSamplesToFilter:=cal_mva_nSamplesToFilter,
			nWorkArray_SIZEOF:=cal_mva_nWorkArray_SIZEOF),
		(	tTaskCycleTime:=cal_tm_task, 
			tCtrlCycleTime:=cal_tm,
			nSamplesToFilter:=cal_mva_nSamplesToFilter,
			nWorkArray_SIZEOF:=cal_mva_nWorkArray_SIZEOF)
	];
	fb_cal_mva	:	ARRAY[1..4] OF FB_CTRL_MOVING_AVERAGE := [ 
		(eMode:=cal_emode), 
		(eMode:=cal_emode), 
		(eMode:=cal_emode), 
		(eMode:=cal_emode)];
	cal_mva_mbs :	ARRAY[1..4] OF LREAL;

	// more common cal vars		
	cal_10v_dcoffset: ARRAY[1..4] OF LREAL;
	cal_ii: INT;
	cal_diff: ARRAY[1..4] OF LREAL;
	cal_frac: ARRAY[1..4] OF LREAL;
	
END_VAR

VAR CONSTANT
	cal_mva_nSamplesToFilter : UINT := 40;
	cal_mva_nWorkArray_SIZEOF: UINT := 400;
END_VAR


// adjust for test signals

IF test_input THEN
	G_PARAMS.A_FLOW_MAX 		:=10.0;
	G_PARAMS.D_FLOW_MAX			:=10.0;
	G_PARAMS.E_FLOW_MAX			:=10.0;
	G_PARAMS.AC_FLOW_MAX		:=10.0;
	
	G_PARAMS.A_FLOW_MIN 		:=0.0;
	G_PARAMS.D_FLOW_MIN			:=0.0;
	G_PARAMS.E_FLOW_MIN			:=0.0;
	G_PARAMS.AC_FLOW_MIN		:=0.0;
END_IF
//
// BEGIN PRODUCE THE DATA
//
// XMEAS values will come from the external TESIM program using ADS


//
// BEGIN WRITE SIGNALS to OUTPUTS
//
// VOLTAGES
XMEAS_IO_VOUT[XMEAS_IO_IDX.A_FLOW]		:= pv_float_to_dac(pv:=XMEAS[XMEAS_IDX.A_FLOW],		pv_max:=G_PARAMS.A_FLOW_MAX, pv_min:=G_PARAMS.A_FLOW_MIN, dac_max:=VOUT_WD_MAX, dac_min:=0);
XMEAS_IO_VOUT[XMEAS_IO_IDX.D_FLOW]		:= pv_float_to_dac(pv:=XMEAS[XMEAS_IDX.D_FLOW],		pv_max:=G_PARAMS.D_FLOW_MAX, pv_min:=G_PARAMS.D_FLOW_MIN, dac_max:=VOUT_WD_MAX, dac_min:=0);
XMEAS_IO_VOUT[XMEAS_IO_IDX.E_FLOW]		:= pv_float_to_dac(pv:=XMEAS[XMEAS_IDX.E_FLOW],		pv_max:=G_PARAMS.E_FLOW_MAX, pv_min:=G_PARAMS.E_FLOW_MIN, dac_max:=VOUT_WD_MAX, dac_min:=0);
XMEAS_IO_VOUT[XMEAS_IO_IDX.AC_FLOW]	:= pv_float_to_dac(pv:=XMEAS[XMEAS_IDX.AC_FLOW],	pv_max:=G_PARAMS.AC_FLOW_MAX, pv_min:=G_PARAMS.AC_FLOW_MIN, dac_max:=VOUT_WD_MAX, dac_min:=0);

//
// BEGIN MODBUS POLLING SEGMENT from the GATEWAY
//
fbReadMB(addrs := mbAddrs );

// poll modbus registers
G_IO.MBS_XMEAS_RAW[XMEAS_MBS_IDX.A_FLOW] := fbReadMB.registerValues[XMEAS_MBS_IDX.A_FLOW] + MBS_XMEAS_CAL_OFFSET[1];
G_IO.MBS_XMEAS_RAW[XMEAS_MBS_IDX.D_FLOW] := fbReadMB.registerValues[XMEAS_MBS_IDX.D_FLOW]+ MBS_XMEAS_CAL_OFFSET[2];
G_IO.MBS_XMEAS_RAW[XMEAS_MBS_IDX.E_FLOW] := fbReadMB.registerValues[XMEAS_MBS_IDX.E_FLOW] + MBS_XMEAS_CAL_OFFSET[3];
G_IO.MBS_XMEAS_RAW[XMEAS_MBS_IDX.AC_FLOW] := fbReadMB.registerValues[XMEAS_MBS_IDX.AC_FLOW] + MBS_XMEAS_CAL_OFFSET[4];

// convert raw modbus signals to process signals
G_IO.MBS_XMEAS[XMEAS_MBS_IDX.A_FLOW]	:=	LREAL_TO_REAL(adc_to_float_pv(G_IO.MBS_XMEAS_RAW[XMEAS_MBS_IDX.A_FLOW],		pv_max:=G_PARAMS.A_FLOW_MAX, 		pv_min:=G_PARAMS.A_FLOW_MIN, 	i_max:=G_PARAMS.VOUT_MAX, i_min:=G_PARAMS.VOUT_MIN));
G_IO.MBS_XMEAS[XMEAS_MBS_IDX.D_FLOW]	:=	LREAL_TO_REAL(adc_to_float_pv(G_IO.MBS_XMEAS_RAW[XMEAS_MBS_IDX.D_FLOW],		pv_max:=G_PARAMS.D_FLOW_MAX, 		pv_min:=G_PARAMS.D_FLOW_MIN, 	i_max:=G_PARAMS.VOUT_MAX, i_min:=G_PARAMS.VOUT_MIN));
G_IO.MBS_XMEAS[XMEAS_MBS_IDX.E_FLOW]	:=	LREAL_TO_REAL(adc_to_float_pv(G_IO.MBS_XMEAS_RAW[XMEAS_MBS_IDX.E_FLOW],		pv_max:=G_PARAMS.E_FLOW_MAX, 		pv_min:=G_PARAMS.E_FLOW_MIN, 	i_max:=G_PARAMS.VOUT_MAX, i_min:=G_PARAMS.VOUT_MIN));
G_IO.MBS_XMEAS[XMEAS_MBS_IDX.AC_FLOW]	:=	LREAL_TO_REAL(adc_to_float_pv(G_IO.MBS_XMEAS_RAW[XMEAS_MBS_IDX.AC_FLOW],	pv_max:=G_PARAMS.AC_FLOW_MAX, 	pv_min:=G_PARAMS.AC_FLOW_MIN, i_max:=G_PARAMS.VOUT_MAX, i_min:=G_PARAMS.VOUT_MIN));


//
// END MODBUS POLLING SEGMENT from the GATEWAY
//




		
// CALIBRATION SECTION
IF cal_override THEN
	FOR cal_ii := 1 TO 4 DO
		CASE cal_ii OF
			1:
			G_IO.XMEAS[XMEAS_IDX.A_FLOW]:=0.5;
			2:
			G_IO.XMEAS[XMEAS_IDX.D_FLOW] := 1500;
			3:
			G_IO.XMEAS[XMEAS_IDX.E_FLOW] := 1500;
			4:
			G_IO.XMEAS[XMEAS_IDX.AC_FLOW] := 2500;
		END_CASE
	END_FOR
END_IF
IF cal_emode=eCTRL_MODE_ACTIVE THEN
	FOR cal_ii := 1 TO 4 DO
		CASE cal_ii OF
			1:
			cal_pv_mbs[cal_ii] := G_IO.MBS_XMEAS[XMEAS_MBS_IDX.A_FLOW];
			cal_pv[cal_ii] := G_IO.XMEAS[XMEAS_IDX.A_FLOW];
			2:
			cal_pv_mbs[cal_ii] := G_IO.MBS_XMEAS[XMEAS_MBS_IDX.D_FLOW];
			cal_pv[cal_ii] := G_IO.XMEAS[XMEAS_IDX.D_FLOW];
			3:
			cal_pv_mbs[cal_ii] := G_IO.MBS_XMEAS[XMEAS_MBS_IDX.E_FLOW];
			cal_pv[cal_ii] := G_IO.XMEAS[XMEAS_IDX.E_FLOW];
			4:
			cal_pv_mbs[cal_ii] := G_IO.MBS_XMEAS[XMEAS_MBS_IDX.AC_FLOW];
			cal_pv[cal_ii] := G_IO.XMEAS[XMEAS_IDX.AC_FLOW];
		END_CASE
	
		// calculate moving average
		cal_mva_st[cal_ii].pWorkArray_ADR	:= ADR(cal_mva_work[cal_ii]);
		fb_cal_mva[cal_ii].fIn := cal_pv_mbs[cal_ii];
		fb_cal_mva[cal_ii](stParams:=cal_mva_st[cal_ii], eMode:=cal_emode);
		cal_mva_mbs[cal_ii] := fb_cal_mva[cal_ii].fOut;	
		
		// calculate dc offset
		IF ABS(cal_pv[cal_ii]) > 0.0 THEN
			cal_diff[cal_ii]:=cal_mva_mbs[cal_ii]-cal_pv[cal_ii];
			cal_frac[cal_ii]:=cal_diff[cal_ii]/cal_pv[cal_ii];
			cal_10v_dcoffset[cal_ii] := 10.0*cal_frac[cal_ii];
		END_IF
		
	END_FOR	
END_IF

END_PROGRAM

// ---- GlobalTextList.TcGTLO
TEXTLIST GlobalTextList
  32 = '"Setpoint"'
  58 = '%0.0f $/hr'
  51 = '%0.0f cmh'
  50 = '%0.0f kmh'
  45 = '%0.0f kPa'
  44 = '%0.1f'
  35 = '%0.1f %'
  37 = '%0.1f C'
  54 = '%0.1f cmh'
  59 = '%0.1f kgph'
  60 = '%0.1f kscmh'
  5 = '%0.3f'
  25 = '%0.3f %'
  36 = '%0.3f C'
  27 = '%0.3f cu. m/h'
  28 = '%0.3f deg'
  26 = '%0.3f deg C'
  21 = '%0.3f kg/h'
  22 = '%0.3f kPa'
  24 = '%0.3f kPa %'
  23 = '%0.3f kPa \\%'
  20 = '%0.3f kscmh'
  29 = '%0.3f kW'
  34 = '%0.3f \\%'
  31 = '%0.3f,%0.3f,%0.3f,%0.3f,%0.3f,%0.3f,%0.3f,%0.3f'
  30 = '%0.3f,%0.3f,%0.3f,%0.3f,%0.3f,%0.3f,%0.3f,%0.3f,\\'
  1 = '%G_IO.XMEAS[8]'
  92 = '%i'
  4 = '%s'
  67 = '0'
  68 = '1'
  77 = '10'
  78 = '11'
  79 = '12'
  80 = '13'
  81 = '14'
  82 = '15'
  83 = '16'
  85 = '17'
  86 = '18'
  87 = '19'
  69 = '2'
  88 = '20'
  70 = '3'
  71 = '4'
  72 = '5'
  73 = '6'
  74 = '7'
  75 = '8'
  76 = '9'
  2 = '=G_IO.XMEAS[8]'
  61 = 'Chemical Reactor Process,  Operating Time: %0.2f'
  62 = 'Chemical Reactor Process, Operating Time: %0.2f'
  63 = 'Chemical Reactor Process, Operating Time: %0.3f'
  64 = 'Chemical Reactor Process, Running Time: %0.3f hours'
  47 = 'Condenser'
  57 = 'Cost'
  65 = 'Disturbances'
  53 = 'Flow'
  3 = 'ggggg'
  0 = 'G_IO.XMEAS[8]'
  66 = 'IDV'
  84 = 'IDV %i'
  97 = 'IDVs'
  12 = 'LEVEL'
  39 = 'Level'
  96 = 'MODE'
  18 = 'Name'
  94 = 'NET'
  89 = 'NET TYPE'
  91 = 'NETT'
  90 = 'NETTYPE'
  56 = 'Pct G'
  42 = 'Press.'
  17 = 'PRESS. (kPa)'
  13 = 'PRESSURE'
  15 = 'PRESSURE (kPa)'
  16 = 'PRESSURE \\n(kPa)'
  49 = 'Prod.'
  52 = 'Product'
  55 = 'Quality'
  6 = 'REACTOR'
  38 = 'Reactor'
  9 = 'REACTOR:'
  7 = 'SEPARATOR'
  46 = 'Separator'
  10 = 'SEPARATOR:'
  33 = 'Setpoint'
  8 = 'STRIPPER'
  48 = 'Stripper'
  11 = 'STRIPPER:'
  40 = 'Temp'
  14 = 'TEMP (C)'
  41 = 'Temp (C)'
  43 = 'Temp.'
  95 = 'TYPE'
  93 = 'USE'
  19 = 'Value'
END_TEXTLIST

// ---- VISUs/TankView.TcVIS
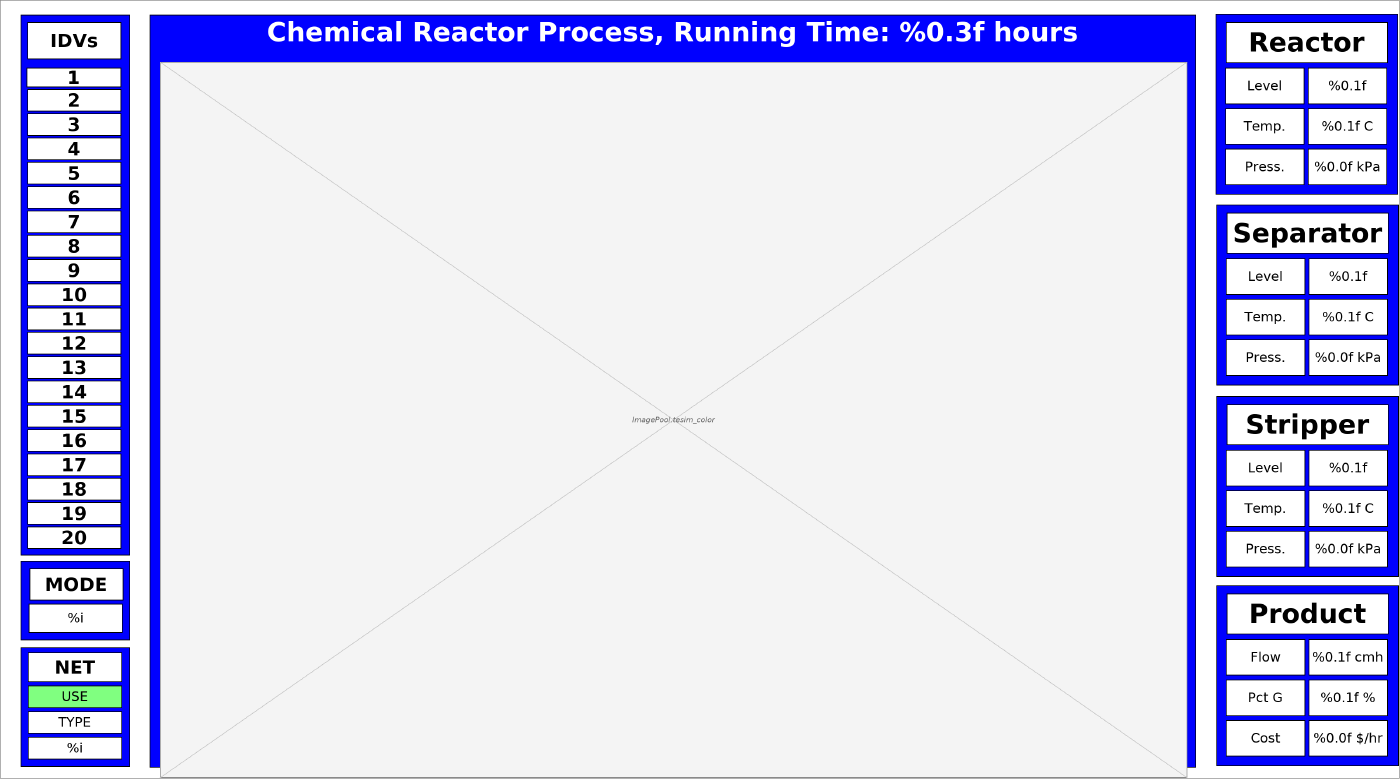
VISUALIZATION TankView  // 1899x1058
    Rectangle (203,20 1419x1022), "Chemical Reactor Process, Running Time: %0.3f hours", text variable: OPTIME
    Rectangle (1649,19 247x245)
    Rectangle (1663,30 219x55), "Reactor"
    Rectangle (1774,92 107x49), "%0.1f", text variable: G_IO.XMEAS[8]
    Rectangle (1774,147 107x49), "%0.1f C", text variable: G_IO.XMEAS[9]
    Rectangle (1774,202 107x49), "%0.0f kPa", text variable: G_IO.XMEAS[7]
    Rectangle (1662,92 107x49), "Level"
    Rectangle (1662,147 107x49), "Temp."
    Rectangle (1662,202 107x49), "Press."
    Rectangle (1650,278 247x245)
    Rectangle (1664,289 219x55), "Separator"
    Rectangle (1775,351 107x49), "%0.1f", text variable: G_IO.XMEAS[12]
    Rectangle (1775,406 107x49), "%0.1f C", text variable: G_IO.XMEAS[11]
    Rectangle (1775,461 107x49), "%0.0f kPa", text variable: G_IO.XMEAS[13]
    Rectangle (1663,351 107x49), "Level"
    Rectangle (1663,406 107x49), "Temp."
    Rectangle (1663,461 107x49), "Press."
    Rectangle (1650,538 247x245)
    Rectangle (1664,549 219x55), "Stripper"
    Rectangle (1775,611 107x49), "%0.1f", text variable: G_IO.XMEAS[15]
    Rectangle (1775,666 107x49), "%0.1f C", text variable: G_IO.XMEAS[18]
    Rectangle (1775,721 107x49), "%0.0f kPa", text variable: G_IO.XMEAS[16]
    Rectangle (1663,611 107x49), "Level"
    Rectangle (1663,666 107x49), "Temp."
    Rectangle (1663,721 107x49), "Press."
    Rectangle (1650,795 247x245)
    Rectangle (1664,806 219x55), "Product"
    Rectangle (1775,868 107x49), "%0.1f cmh", text variable: G_IO.XMEAS[17]
    Rectangle (1775,923 107x49), "%0.1f %", text variable: G_IO.XMEAS[40]
    Rectangle (1775,978 107x49), "%0.0f $/hr", text variable: G_IO.COST
    Rectangle (1663,868 107x49), "Flow"
    Rectangle (1663,923 107x49), "Pct G"
    Rectangle (1663,978 107x49), "Cost"
    Rectangle (221,200 190x49), "%0.3f kscmh", text variable: G_IO.XMEAS[1]
    Rectangle (221,364 192x49), "%0.1f kgph", text variable: G_IO.XMEAS[2]
    Rectangle (221,515 202x49), "%0.1f kgph", text variable: G_IO.XMEAS[3]
    Rectangle (460,915 200x49), "%0.3f kscmh", text variable: G_IO.XMEAS[4]
    Rectangle (28,20 148x734)
    Rectangle (37,30 127x50), "IDVs"
    Rectangle (36,92 128x26), "1", invisible if: Not(udint_to_bool(IDV[1]))
    Rectangle (37,121 127x30), "2", invisible if: Not(udint_to_bool(IDV[2]))
    Rectangle (37,154 127x30), "3", invisible if: Not(udint_to_bool(IDV[3]))
    Rectangle (37,187 127x30), "4", invisible if: Not(udint_to_bool(IDV[4]))
    Rectangle (37,220 127x30), "5", invisible if: Not(udint_to_bool(IDV[5]))
    Rectangle (37,253 127x30), "6", invisible if: Not(udint_to_bool(IDV[6]))
    Rectangle (37,286 127x30), "7", invisible if: Not(udint_to_bool(IDV[7]))
    Rectangle (37,319 127x30), "8", invisible if: Not(udint_to_bool(IDV[8]))
    Rectangle (37,352 127x30), "9", invisible if: Not(udint_to_bool(IDV[9]))
    Rectangle (37,385 127x30), "10", invisible if: Not(udint_to_bool(IDV[10]))
    Rectangle (37,418 127x30), "11", invisible if: Not(udint_to_bool(IDV[11]))
    Rectangle (37,451 127x30), "12", invisible if: Not(udint_to_bool(IDV[12]))
    Rectangle (37,484 127x30), "13", invisible if: Not(udint_to_bool(IDV[13]))
    Rectangle (37,517 127x30), "14", invisible if: Not(udint_to_bool(IDV[14]))
    Rectangle (37,550 127x30), "15", invisible if: Not(udint_to_bool(IDV[15]))
    Rectangle (37,583 127x30), "16", invisible if: Not(udint_to_bool(IDV[16]))
    Rectangle (37,616 127x30), "17", invisible if: Not(udint_to_bool(IDV[17]))
    Rectangle (37,649 127x30), "18", invisible if: Not(udint_to_bool(IDV[18]))
    Rectangle (37,682 127x30), "19", invisible if: Not(udint_to_bool(IDV[19]))
    Rectangle (37,715 127x30), "20", invisible if: Not(udint_to_bool(G_IO.IDV[20]))
    Rectangle (28,879 148x162)
    Rectangle (38,886 127x40), "NET"
    Rectangle (38,1001 127x30), "%i", text variable: NET_TYPE
    Rectangle (38,931 127x30), "USE", invisible if: Not(GO)
    Rectangle (38,966 127x30), "TYPE"
    Rectangle (28,762 148x107)
    Rectangle (40,772 127x43), "MODE"
    Rectangle (39,820 127x39), "%i", text variable: MODE
    Image (217,84 1393x972), image: ImagePool.tesim_color
END_VISUALIZATION
